LIN {X -0.248,Y -541.721,Z 1405.628,A 0.000,B 0.000,C 90.000,E1 148.997} C_DIS
LIN {X -0.026,Y -544.533,Z 1405.623,A 0.000,B 0.000,C 90.000,E1 148.122} C_DIS
LIN {X 0.196,Y -546.222,Z 1405.620,A 0.000,B 0.000,C 90.000,E1 147.533} C_DIS
LIN {X 0.004,Y -548.398,Z 1405.615,A 0.000,B 0.000,C 90.000,E1 146.707} C_DIS
LIN {X -0.112,Y -550.816,Z 1405.609,A 0.000,B 0.000,C 90.000,E1 145.595} C_DIS
LIN {X -0.256,Y -552.252,Z 1405.604,A 0.000,B 0.000,C 90.000,E1 144.769} C_DIS
LIN {X -0.066,Y -553.322,Z 1405.599,A 0.000,B 0.000,C 90.000,E1 143.909} C_DIS
LIN {X 0.212,Y -554.490,Z 1405.593,A 0.000,B 0.000,C 90.000,E1 142.763} C_DIS
LIN {X 0.069,Y -555.501,Z 1405.587,A 0.000,B 0.000,C 90.000,E1 141.662} C_DIS
LIN {X 0.018,Y -556.739,Z 1405.579,A 0.000,B 0.000,C 90.000,E1 140.275} C_DIS
LIN {X -0.102,Y -557.519,Z 1405.573,A 0.000,B 0.000,C 90.000,E1 139.175} C_DIS
LIN {X -0.196,Y -558.310,Z 1405.565,A 0.000,B 0.000,C 90.000,E1 137.796} C_DIS
LIN {X 0.032,Y -558.832,Z 1405.559,A 0.000,B 0.000,C 90.000,E1 136.662} C_DIS
LIN {X -0.046,Y -559.385,Z 1405.552,A 0.000,B 0.000,C 90.000,E1 135.283} C_DIS
LIN {X -0.192,Y -559.704,Z 1405.545,A 0.000,B 0.000,C 90.000,E1 134.190} C_DIS
LIN {X 0.136,Y -560.065,Z 1405.538,A 0.000,B 0.000,C 90.000,E1 132.771} C_DIS
LIN {X 0.008,Y -560.188,Z 1405.532,A 0.000,B 0.000,C 90.000,E1 131.676} C_DIS
LIN {X 0.139,Y -560.368,Z 1405.521,A 0.000,B 0.000,C 90.000,E1 129.725} C_DIS
LIN {X -0.174,Y -560.676,Z 1405.512,A 0.000,B 0.000,C 90.000,E1 128.096} C_DIS
LIN {X -0.144,Y -560.829,Z 1405.504,A 0.000,B 0.000,C 90.000,E1 126.710} C_DIS
LIN {X 0.003,Y -560.849,Z 1405.496,A 0.000,B 0.000,C 90.000,E1 125.311} C_DIS
LIN {X -0.005,Y -561.268,Z 1405.481,A 0.000,B 0.000,C 90.000,E1 122.546} C_DIS
LIN {X 0.083,Y -561.611,Z 1405.479,A 0.000,B 0.000,C 90.000,E1 122.260} C_DIS
LIN {X -0.232,Y -561.927,Z 1405.477,A 0.000,B 0.000,C 90.000,E1 121.878} C_DIS
LIN {X -0.040,Y -562.328,Z 1405.476,A 0.000,B 0.000,C 90.000,E1 121.720} C_DIS
LIN {X -0.254,Y -563.108,Z 1405.474,A 0.000,B 0.000,C 90.000,E1 121.258} C_DIS
LIN {X 0.206,Y -564.134,Z 1405.472,A 0.000,B 0.000,C 90.000,E1 121.003} C_DIS
LIN {X -0.097,Y -566.068,Z 1405.472,A 0.000,B 0.000,C 90.000,E1 120.924} C_DIS
LIN {X -0.002,Y -567.840,Z 1405.471,A 0.000,B 0.000,C 90.000,E1 120.846} C_DIS
LIN {X 0.227,Y -573.827,Z 1405.471,A 0.000,B 0.000,C 90.000,E1 120.669} C_DIS
LIN {X 0.258,Y -579.247,Z 1405.470,A 0.000,B 0.000,C 90.000,E1 120.590} C_DIS
LIN {X 0.183,Y -581.728,Z 1405.470,A 0.000,B 0.000,C 90.000,E1 120.541} C_DIS
LIN {X 0.143,Y -584.144,Z 1405.469,A 0.000,B 0.000,C 90.000,E1 120.463} C_DIS
LIN {X 0.234,Y -586.696,Z 1405.469,A 0.000,B 0.000,C 90.000,E1 120.335} C_DIS
LIN {X -0.041,Y -589.555,Z 1405.468,A 0.000,B 0.000,C 90.000,E1 120.207} C_DIS
LIN {X 0.287,Y -592.453,Z 1405.467,A 0.000,B 0.000,C 90.000,E1 120.001} C_DIS
LIN {X 0.078,Y -597.897,Z 1405.465,A 0.000,B 0.000,C 90.000,E1 119.617} C_DIS
LIN {X 0.189,Y -603.137,Z 1405.462,A 0.000,B 0.000,C 90.000,E1 119.155} C_DIS
LIN {X -0.118,Y -606.860,Z 1405.460,A 0.000,B 0.000,C 90.000,E1 118.821} C_DIS
LIN {X -0.111,Y -609.008,Z 1405.459,A 0.000,B 0.000,C 90.000,E1 118.565} C_DIS
LIN {X 0.109,Y -612.046,Z 1405.457,A 0.000,B 0.000,C 90.000,E1 118.153} C_DIS
LIN {X 0.041,Y -615.591,Z 1405.454,A 0.000,B 0.000,C 90.000,E1 117.641} C_DIS
LIN {X -0.008,Y -619.104,Z 1405.450,A 0.000,B 0.000,C 90.000,E1 117.001} C_DIS
LIN {X -0.015,Y -619.633,Z 1405.449,A 0.000,B 0.000,C 90.000,E1 116.873} C_DIS
LIN {X -0.036,Y -621.269,Z 1405.445,A 0.000,B 0.000,C 90.000,E1 116.104} C_DIS
LIN {X -0.040,Y -621.342,Z 1405.444,A 0.000,B 0.000,C 90.000,E1 115.848} C_DIS
LIN {X -0.042,Y -621.209,Z 1405.442,A 0.000,B 0.000,C 90.000,E1 115.591} C_DIS
LIN {X -0.044,Y -620.763,Z 1405.441,A 0.000,B 0.000,C 90.000,E1 115.335} C_DIS
LIN {X -0.053,Y -618.848,Z 1405.438,A 0.000,B 0.000,C 90.000,E1 114.823} C_DIS
LIN {X -0.062,Y -616.821,Z 1405.437,A 0.000,B 0.000,C 90.000,E1 114.567} C_DIS
LIN {X 0.030,Y -614.783,Z 1405.435,A 0.000,B 0.000,C 90.000,E1 114.259} C_DIS
LIN {X 0.020,Y -613.342,Z 1405.434,A 0.000,B 0.000,C 90.000,E1 114.131} C_DIS
LIN {X -0.037,Y -606.794,Z 1405.432,A 0.000,B 0.000,C 90.000,E1 113.695} C_DIS
LIN {X 0.065,Y -599.335,Z 1405.430,A 0.000,B 0.000,C 90.000,E1 113.334} C_DIS
LIN {X -0.118,Y -589.005,Z 1405.427,A 0.000,B 0.000,C 90.000,E1 112.950} C_DIS
LIN {X 0.105,Y -585.189,Z 1405.427,A 0.000,B 0.000,C 90.000,E1 112.770} C_DIS
LIN {X 0.059,Y -585.235,Z 1405.427,A 0.000,B 0.000,C 90.000,E1 112.770} C_DIS
LIN {X -0.328,Y -588.195,Z 1405.425,A 0.000,B 0.000,C 90.000,E1 112.589} C_DIS
LIN {X 0.216,Y -595.378,Z 1405.423,A 0.000,B 0.000,C 90.000,E1 112.078} C_DIS
LIN {X -0.256,Y -601.161,Z 1405.421,A 0.000,B 0.000,C 90.000,E1 111.716} C_DIS
LIN {X 0.185,Y -605.437,Z 1405.419,A 0.000,B 0.000,C 90.000,E1 111.354} C_DIS
LIN {X 0.068,Y -610.886,Z 1405.416,A 0.000,B 0.000,C 90.000,E1 110.918} C_DIS
LIN {X 0.296,Y -617.284,Z 1405.413,A 0.000,B 0.000,C 90.000,E1 110.301} C_DIS
LIN {X 0.233,Y -621.031,Z 1405.411,A 0.000,B 0.000,C 90.000,E1 109.939} C_DIS
LIN {X 0.039,Y -625.525,Z 1405.408,A 0.000,B 0.000,C 90.000,E1 109.450} C_DIS
LIN {X -0.190,Y -629.572,Z 1405.405,A 0.000,B 0.000,C 90.000,E1 108.960} C_DIS
LIN {X 0.021,Y -634.903,Z 1405.401,A 0.000,B 0.000,C 90.000,E1 108.181} C_DIS
LIN {X -0.327,Y -638.717,Z 1405.398,A 0.000,B 0.000,C 90.000,E1 107.583} C_DIS
LIN {X -0.030,Y -642.239,Z 1405.393,A 0.000,B 0.000,C 90.000,E1 106.804} C_DIS
LIN {X -0.166,Y -643.953,Z 1405.391,A 0.000,B 0.000,C 90.000,E1 106.315} C_DIS
LIN {X 0.299,Y -644.698,Z 1405.389,A 0.000,B 0.000,C 90.000,E1 106.024} C_DIS
LIN {X 0.003,Y -645.737,Z 1405.386,A 0.000,B 0.000,C 90.000,E1 105.552} C_DIS
LIN {X 0.222,Y -647.242,Z 1405.381,A 0.000,B 0.000,C 90.000,E1 104.537} C_DIS
LIN {X -0.195,Y -648.196,Z 1405.377,A 0.000,B 0.000,C 90.000,E1 103.828} C_DIS
LIN {X 0.027,Y -648.755,Z 1405.373,A 0.000,B 0.000,C 90.000,E1 103.063} C_DIS
LIN {X -0.243,Y -648.886,Z 1405.370,A 0.000,B 0.000,C 90.000,E1 102.591} C_DIS
LIN {X -0.016,Y -648.656,Z 1405.366,A 0.000,B 0.000,C 90.000,E1 101.827} C_DIS
LIN {X 0.343,Y -648.336,Z 1405.363,A 0.000,B 0.000,C 90.000,E1 101.299} C_DIS
LIN {X -0.060,Y -647.747,Z 1405.360,A 0.000,B 0.000,C 90.000,E1 100.838} C_DIS
LIN {X 0.293,Y -646.917,Z 1405.357,A 0.000,B 0.000,C 90.000,E1 100.310} C_DIS
LIN {X -0.259,Y -645.272,Z 1405.353,A 0.000,B 0.000,C 90.000,E1 99.613} C_DIS
LIN {X -0.033,Y -643.887,Z 1405.351,A 0.000,B 0.000,C 90.000,E1 99.095} C_DIS
LIN {X 0.286,Y -642.274,Z 1405.348,A 0.000,B 0.000,C 90.000,E1 98.568} C_DIS
LIN {X -0.140,Y -640.471,Z 1405.345,A 0.000,B 0.000,C 90.000,E1 98.106} C_DIS
LIN {X -0.120,Y -637.221,Z 1405.341,A 0.000,B 0.000,C 90.000,E1 97.352} C_DIS
LIN {X -0.075,Y -634.206,Z 1405.337,A 0.000,B 0.000,C 90.000,E1 96.720} C_DIS
LIN {X 0.080,Y -631.519,Z 1405.335,A 0.000,B 0.000,C 90.000,E1 96.201} C_DIS
LIN {X -0.149,Y -626.443,Z 1405.330,A 0.000,B 0.000,C 90.000,E1 95.334} C_DIS
LIN {X -0.198,Y -622.212,Z 1405.326,A 0.000,B 0.000,C 90.000,E1 94.702} C_DIS
LIN {X -0.176,Y -618.355,Z 1405.323,A 0.000,B 0.000,C 90.000,E1 94.188} C_DIS
LIN {X -0.092,Y -612.452,Z 1405.320,A 0.000,B 0.000,C 90.000,E1 93.555} C_DIS
LIN {X 0.056,Y -604.236,Z 1405.316,A 0.000,B 0.000,C 90.000,E1 92.808} C_DIS
LIN {X -0.056,Y -597.375,Z 1405.313,A 0.000,B 0.000,C 90.000,E1 92.236} C_DIS
LIN {X 0.161,Y -590.138,Z 1405.309,A 0.000,B 0.000,C 90.000,E1 91.661} C_DIS
LIN {X -0.180,Y -581.695,Z 1405.307,A 0.000,B 0.000,C 90.000,E1 91.203} C_DIS
LIN {X -0.243,Y -578.344,Z 1405.306,A 0.000,B 0.000,C 90.000,E1 91.031} C_DIS
LIN {X 0.048,Y -577.150,Z 1405.305,A 0.000,B 0.000,C 90.000,E1 90.917} C_DIS
LIN {X -0.255,Y -576.182,Z 1405.305,A 0.000,B 0.000,C 90.000,E1 90.859} C_DIS
LIN {X -0.076,Y -574.207,Z 1405.304,A 0.000,B 0.000,C 90.000,E1 90.688} C_DIS
LIN {X 0.146,Y -573.809,Z 1405.303,A 0.000,B 0.000,C 90.000,E1 90.573} C_DIS
LIN {X -0.068,Y -573.399,Z 1405.303,A 0.000,B 0.000,C 90.000,E1 90.458} C_DIS
LIN {X -0.139,Y -573.123,Z 1405.300,A 0.000,B 0.000,C 90.000,E1 90.057} C_DIS
LIN {X -0.252,Y -573.569,Z 1405.296,A 0.000,B 0.000,C 90.000,E1 89.255} C_DIS
LIN {X -0.237,Y -574.603,Z 1405.290,A 0.000,B 0.000,C 90.000,E1 88.165} C_DIS
LIN {X 0.097,Y -576.049,Z 1405.281,A 0.000,B 0.000,C 90.000,E1 86.502} C_DIS
LIN {X 0.260,Y -578.153,Z 1405.269,A 0.000,B 0.000,C 90.000,E1 84.318} C_DIS
LIN {X 0.173,Y -579.997,Z 1405.260,A 0.000,B 0.000,C 90.000,E1 82.704} C_DIS
LIN {X 0.081,Y -582.504,Z 1405.248,A 0.000,B 0.000,C 90.000,E1 80.557} C_DIS
LIN {X 0.256,Y -584.296,Z 1405.239,A 0.000,B 0.000,C 90.000,E1 78.926} C_DIS
LIN {X 0.209,Y -585.615,Z 1405.231,A 0.000,B 0.000,C 90.000,E1 77.589} C_DIS
LIN {X -0.209,Y -587.158,Z 1405.221,A 0.000,B 0.000,C 90.000,E1 75.755} C_DIS
LIN {X 0.051,Y -588.113,Z 1405.213,A 0.000,B 0.000,C 90.000,E1 74.393} C_DIS
LIN {X 0.169,Y -588.956,Z 1405.204,A 0.000,B 0.000,C 90.000,E1 72.779} C_DIS
LIN {X 0.057,Y -589.735,Z 1405.197,A 0.000,B 0.000,C 90.000,E1 71.456} C_DIS
LIN {X 0.271,Y -590.290,Z 1405.191,A 0.000,B 0.000,C 90.000,E1 70.369} C_DIS
LIN {X 0.254,Y -591.216,Z 1405.182,A 0.000,B 0.000,C 90.000,E1 68.773} C_DIS
LIN {X -0.293,Y -592.162,Z 1405.173,A 0.000,B 0.000,C 90.000,E1 67.230} C_DIS
LIN {X 0.047,Y -593.134,Z 1405.166,A 0.000,B 0.000,C 90.000,E1 65.869} C_DIS
LIN {X -0.174,Y -594.804,Z 1405.154,A 0.000,B 0.000,C 90.000,E1 63.768} C_DIS
LIN {X -0.003,Y -595.667,Z 1405.148,A 0.000,B 0.000,C 90.000,E1 62.692} C_DIS
LIN {X -0.251,Y -596.932,Z 1405.140,A 0.000,B 0.000,C 90.000,E1 61.129} C_DIS
LIN {X -0.090,Y -598.138,Z 1405.132,A 0.000,B 0.000,C 90.000,E1 59.793} C_DIS
LIN {X 0.245,Y -599.835,Z 1405.122,A 0.000,B 0.000,C 90.000,E1 57.916} C_DIS
LIN {X -0.046,Y -601.029,Z 1405.115,A 0.000,B 0.000,C 90.000,E1 56.628} C_DIS
LIN {X 0.169,Y -602.724,Z 1405.104,A 0.000,B 0.000,C 90.000,E1 54.769} C_DIS
LIN {X 0.015,Y -604.096,Z 1405.096,A 0.000,B 0.000,C 90.000,E1 53.210} C_DIS
LIN {X -0.011,Y -605.038,Z 1405.088,A 0.000,B 0.000,C 90.000,E1 51.904} C_DIS
LIN {X -0.285,Y -605.755,Z 1405.083,A 0.000,B 0.000,C 90.000,E1 50.884} C_DIS
LIN {X 0.097,Y -606.454,Z 1405.075,A 0.000,B 0.000,C 90.000,E1 49.542} C_DIS
LIN {X 0.224,Y -606.791,Z 1405.070,A 0.000,B 0.000,C 90.000,E1 48.485} C_DIS
LIN {X -0.098,Y -606.994,Z 1405.064,A 0.000,B 0.000,C 90.000,E1 47.472} C_DIS
LIN {X 0.253,Y -607.092,Z 1405.057,A 0.000,B 0.000,C 90.000,E1 46.134} C_DIS
LIN {X 0.170,Y -606.960,Z 1405.049,A 0.000,B 0.000,C 90.000,E1 44.838} C_DIS
LIN {X -0.396,Y -606.798,Z 1405.045,A 0.000,B 0.000,C 90.000,E1 44.109} C_DIS
LIN {X -0.049,Y -606.219,Z 1405.038,A 0.000,B 0.000,C 90.000,E1 42.771} C_DIS
LIN {X -0.376,Y -605.679,Z 1405.032,A 0.000,B 0.000,C 90.000,E1 41.757} C_DIS
LIN {X -0.258,Y -604.916,Z 1405.026,A 0.000,B 0.000,C 90.000,E1 40.701} C_DIS
LIN {X -0.151,Y -604.057,Z 1405.020,A 0.000,B 0.000,C 90.000,E1 39.644} C_DIS
LIN {X 0.191,Y -602.658,Z 1405.013,A 0.000,B 0.000,C 90.000,E1 38.302} C_DIS
LIN {X -0.121,Y -601.286,Z 1405.007,A 0.000,B 0.000,C 90.000,E1 37.282} C_DIS
LIN {X 0.028,Y -599.737,Z 1405.001,A 0.000,B 0.000,C 90.000,E1 36.217} C_DIS
LIN {X 0.046,Y -597.330,Z 1404.994,A 0.000,B 0.000,C 90.000,E1 34.898} C_DIS
LIN {X -0.091,Y -595.578,Z 1404.990,A 0.000,B 0.000,C 90.000,E1 34.119} C_DIS
LIN {X 0.136,Y -593.099,Z 1404.984,A 0.000,B 0.000,C 90.000,E1 33.038} C_DIS
LIN {X -0.167,Y -590.165,Z 1404.978,A 0.000,B 0.000,C 90.000,E1 32.005} C_DIS
LIN {X -0.201,Y -587.697,Z 1404.973,A 0.000,B 0.000,C 90.000,E1 31.209} C_DIS
LIN {X 0.039,Y -584.826,Z 1404.969,A 0.000,B 0.000,C 90.000,E1 30.384} C_DIS
LIN {X -0.213,Y -582.703,Z 1404.966,A 0.000,B 0.000,C 90.000,E1 29.873} C_DIS
LIN {X 0.184,Y -579.098,Z 1404.961,A 0.000,B 0.000,C 90.000,E1 29.027} C_DIS
LIN {X 0.029,Y -575.229,Z 1404.957,A 0.000,B 0.000,C 90.000,E1 28.231} C_DIS
LIN {X 0.167,Y -569.424,Z 1404.951,A 0.000,B 0.000,C 90.000,E1 27.129} C_DIS
LIN {X -0.034,Y -563.032,Z 1404.945,A 0.000,B 0.000,C 90.000,E1 26.052} C_DIS
LIN {X 0.128,Y -557.707,Z 1404.940,A 0.000,B 0.000,C 90.000,E1 25.207} C_DIS
LIN {X -0.186,Y -554.901,Z 1404.938,A 0.000,B 0.000,C 90.000,E1 24.823} C_DIS
LIN {X 0.265,Y -549.905,Z 1404.934,A 0.000,B 0.000,C 90.000,E1 24.079} C_DIS
LIN {X -0.089,Y -546.716,Z 1404.932,A 0.000,B 0.000,C 90.000,E1 23.695} C_DIS
LIN {X 0.154,Y -539.977,Z 1404.927,A 0.000,B 0.000,C 90.000,E1 22.823} C_DIS
LIN {X -0.097,Y -535.186,Z 1404.924,A 0.000,B 0.000,C 90.000,E1 22.280} C_DIS
LIN {X -0.121,Y -525.115,Z 1404.917,A 0.000,B 0.000,C 90.000,E1 21.153} C_DIS
LIN {X 0.217,Y -514.660,Z 1404.911,A 0.000,B 0.000,C 90.000,E1 19.993} C_DIS
LIN {X -0.074,Y -503.744,Z 1404.905,A 0.000,B 0.000,C 90.000,E1 18.906} C_DIS
LIN {X 0.113,Y -492.777,Z 1404.899,A 0.000,B 0.000,C 90.000,E1 17.764} C_DIS
LIN {X -0.079,Y -479.251,Z 1404.891,A 0.000,B 0.000,C 90.000,E1 16.386} C_DIS
LIN {X 0.106,Y -465.482,Z 1404.883,A 0.000,B 0.000,C 90.000,E1 14.898} C_DIS
LIN {X 0.055,Y -451.731,Z 1404.875,A 0.000,B 0.000,C 90.000,E1 13.411} C_DIS
LIN {X -0.024,Y -437.847,Z 1404.866,A 0.000,B 0.000,C 90.000,E1 11.883} C_DIS
LIN {X 0.143,Y -417.481,Z 1404.853,A 0.000,B 0.000,C 90.000,E1 9.443} C_DIS
LIN {X -0.048,Y -406.843,Z 1404.845,A 0.000,B 0.000,C 90.000,E1 8.106} C_DIS
LIN {X -0.059,Y -397.404,Z 1404.838,A 0.000,B 0.000,C 90.000,E1 6.891} C_DIS
LIN {X -0.091,Y -393.336,Z 1404.835,A 0.000,B 0.000,C 90.000,E1 6.372} C_DIS
LIN {X -0.063,Y -389.246,Z 1404.832,A 0.000,B 0.000,C 90.000,E1 5.739} C_DIS
LIN {X 0.031,Y -387.720,Z 1404.830,A 0.000,B 0.000,C 90.000,E1 5.391} C_DIS
LIN {X -0.007,Y -387.701,Z 1404.830,A 0.000,B 0.000,C 90.000,E1 5.391} C_DIS
LIN {X -0.180,Y -387.716,Z 1404.829,A 0.000,B 0.000,C 90.000,E1 5.277} C_DIS
LIN {X 0.168,Y -387.721,Z 1404.829,A 0.000,B 0.000,C 90.000,E1 5.220} C_DIS
LIN {X 0.163,Y -389.100,Z 1404.828,A 0.000,B 0.000,C 90.000,E1 4.992} C_DIS
LIN {X -0.132,Y -393.604,Z 1404.825,A 0.000,B 0.000,C 90.000,E1 4.531} C_DIS
LIN {X 0.071,Y -398.766,Z 1404.822,A 0.000,B 0.000,C 90.000,E1 4.012} C_DIS
LIN {X 0.183,Y -403.247,Z 1404.820,A 0.000,B 0.000,C 90.000,E1 3.555} C_DIS
LIN {X 0.078,Y -405.907,Z 1404.818,A 0.000,B 0.000,C 90.000,E1 3.269} C_DIS
LIN {X -0.134,Y -410.707,Z 1404.815,A 0.000,B 0.000,C 90.000,E1 2.694} C_DIS
LIN {X -0.107,Y -416.714,Z 1404.810,A 0.000,B 0.000,C 90.000,E1 1.835} C_DIS
LIN {X -0.025,Y -422.984,Z 1404.804,A 0.000,B 0.000,C 90.000,E1 0.802} C_DIS
LIN {X 0.000,Y -427.486,Z 1404.800,A 0.000,B 0.000,C 90.000,E1 360.000} C_DIS
LIN {X -0.203,Y -430.023,Z 1404.797,A 0.000,B 0.000,C 90.000,E1 359.484} C_DIS
LIN {X -0.131,Y -431.361,Z 1404.795,A 0.000,B 0.000,C 90.000,E1 359.141} C_DIS
LIN {X -0.054,Y -432.419,Z 1404.793,A 0.000,B 0.000,C 90.000,E1 358.797} C_DIS
LIN {X 0.025,Y -433.006,Z 1404.792,A 0.000,B 0.000,C 90.000,E1 358.453} C_DIS
LIN {X 0.121,Y -432.563,Z 1404.790,A 0.000,B 0.000,C 90.000,E1 358.108} C_DIS
LIN {X -0.129,Y -431.791,Z 1404.789,A 0.000,B 0.000,C 90.000,E1 358.051} C_DIS
LIN {X -0.009,Y -430.732,Z 1404.789,A 0.000,B 0.000,C 90.000,E1 357.993} C_DIS
LIN {X 0.095,Y -360.544,Z 1404.787,A 0.000,B 0.000,C 90.000,E1 357.593} C_DIS
LIN {X 0.063,Y -359.781,Z 1404.787,A 0.000,B 0.000,C 90.000,E1 357.593} C_DIS
LIN {X 0.049,Y -359.377,Z 1404.768,A 0.000,B 0.000,C 90.000,E1 354.204} C_DIS
LIN {X -0.057,Y -359.540,Z 1404.726,A 0.000,B 0.000,C 90.000,E1 346.700} C_DIS
LIN {X -0.101,Y -361.978,Z 1404.682,A 0.000,B 0.000,C 90.000,E1 338.827} C_DIS
LIN {X 0.007,Y -365.931,Z 1404.643,A 0.000,B 0.000,C 90.000,E1 331.719} C_DIS
LIN {X -0.235,Y -366.221,Z 1404.641,A 0.000,B 0.000,C 90.000,E1 331.385} C_DIS
LIN {X -0.017,Y -371.299,Z 1404.604,A 0.000,B 0.000,C 90.000,E1 324.689} C_DIS
LIN {X -0.029,Y -371.726,Z 1404.602,A 0.000,B 0.000,C 90.000,E1 324.322} C_DIS
LIN {X 0.051,Y -377.296,Z 1404.567,A 0.000,B 0.000,C 90.000,E1 318.081} C_DIS
LIN {X -0.204,Y -378.205,Z 1404.563,A 0.000,B 0.000,C 90.000,E1 317.391} C_DIS
LIN {X 0.068,Y -383.875,Z 1404.531,A 0.000,B 0.000,C 90.000,E1 311.553} C_DIS
LIN {X 0.117,Y -384.853,Z 1404.527,A 0.000,B 0.000,C 90.000,E1 310.825} C_DIS
LIN {X 0.039,Y -390.546,Z 1404.495,A 0.000,B 0.000,C 90.000,E1 305.105} C_DIS
LIN {X 0.106,Y -391.038,Z 1404.493,A 0.000,B 0.000,C 90.000,E1 304.739} C_DIS
LIN {X -0.048,Y -391.401,Z 1404.491,A 0.000,B 0.000,C 90.000,E1 304.405} C_DIS
LIN {X -0.105,Y -396.764,Z 1404.460,A 0.000,B 0.000,C 90.000,E1 298.743} C_DIS
LIN {X 0.114,Y -397.099,Z 1404.458,A 0.000,B 0.000,C 90.000,E1 298.359} C_DIS
LIN {X -0.101,Y -401.554,Z 1404.427,A 0.000,B 0.000,C 90.000,E1 292.770} C_DIS
LIN {X 0.042,Y -404.617,Z 1404.396,A 0.000,B 0.000,C 90.000,E1 287.166} C_DIS
LIN {X 0.144,Y -404.756,Z 1404.394,A 0.000,B 0.000,C 90.000,E1 286.804} C_DIS
LIN {X 0.142,Y -406.072,Z 1404.365,A 0.000,B 0.000,C 90.000,E1 281.591} C_DIS
LIN {X 0.151,Y -406.113,Z 1404.363,A 0.000,B 0.000,C 90.000,E1 281.243} C_DIS
LIN {X -0.218,Y -405.669,Z 1404.334,A 0.000,B 0.000,C 90.000,E1 276.087} C_DIS
LIN {X 0.191,Y -405.559,Z 1404.332,A 0.000,B 0.000,C 90.000,E1 275.682} C_DIS
LIN {X -0.138,Y -403.525,Z 1404.305,A 0.000,B 0.000,C 90.000,E1 270.859} C_DIS
LIN {X -0.171,Y -403.316,Z 1404.303,A 0.000,B 0.000,C 90.000,E1 270.516} C_DIS
LIN {X 0.018,Y -398.973,Z 1404.272,A 0.000,B 0.000,C 90.000,E1 264.894} C_DIS
LIN {X -0.176,Y -393.145,Z 1404.242,A 0.000,B 0.000,C 90.000,E1 259.634} C_DIS
LIN {X -0.144,Y -392.879,Z 1404.240,A 0.000,B 0.000,C 90.000,E1 259.275} C_DIS
LIN {X -0.121,Y -386.043,Z 1404.213,A 0.000,B 0.000,C 90.000,E1 254.283} C_DIS
LIN {X -0.075,Y -385.314,Z 1404.209,A 0.000,B 0.000,C 90.000,E1 253.559} C_DIS
LIN {X -0.053,Y -384.856,Z 1404.207,A 0.000,B 0.000,C 90.000,E1 253.196} C_DIS
LIN {X 0.049,Y -378.034,Z 1404.183,A 0.000,B 0.000,C 90.000,E1 248.847} C_DIS
LIN {X -0.074,Y -376.287,Z 1404.174,A 0.000,B 0.000,C 90.000,E1 247.411} C_DIS
LIN {X -0.095,Y -375.734,Z 1404.172,A 0.000,B 0.000,C 90.000,E1 247.050} C_DIS
LIN {X 0.009,Y -368.995,Z 1404.150,A 0.000,B 0.000,C 90.000,E1 242.999} C_DIS
LIN {X -0.088,Y -366.137,Z 1404.138,A 0.000,B 0.000,C 90.000,E1 240.795} C_DIS
LIN {X -0.182,Y -359.266,Z 1404.115,A 0.000,B 0.000,C 90.000,E1 236.707} C_DIS
LIN {X 0.044,Y -355.929,Z 1404.100,A 0.000,B 0.000,C 90.000,E1 234.036} C_DIS
LIN {X 0.135,Y -348.858,Z 1404.075,A 0.000,B 0.000,C 90.000,E1 229.461} C_DIS
LIN {X -0.025,Y -346.236,Z 1404.062,A 0.000,B 0.000,C 90.000,E1 227.187} C_DIS
LIN {X 0.098,Y -345.767,Z 1404.060,A 0.000,B 0.000,C 90.000,E1 226.782} C_DIS
LIN {X 0.058,Y -339.037,Z 1404.032,A 0.000,B 0.000,C 90.000,E1 221.757} C_DIS
LIN {X -0.077,Y -336.890,Z 1404.019,A 0.000,B 0.000,C 90.000,E1 219.439} C_DIS
LIN {X -0.060,Y -331.224,Z 1403.991,A 0.000,B 0.000,C 90.000,E1 214.326} C_DIS
LIN {X -0.002,Y -329.324,Z 1403.975,A 0.000,B 0.000,C 90.000,E1 211.544} C_DIS
LIN {X 0.102,Y -326.741,Z 1403.960,A 0.000,B 0.000,C 90.000,E1 208.743} C_DIS
LIN {X 0.049,Y -323.850,Z 1403.929,A 0.000,B 0.000,C 90.000,E1 203.153} C_DIS
LIN {X -0.029,Y -321.117,Z 1403.882,A 0.000,B 0.000,C 90.000,E1 194.717} C_DIS
LIN {X 0.126,Y -320.949,Z 1403.877,A 0.000,B 0.000,C 90.000,E1 193.883} C_DIS
LIN {X -0.095,Y -321.537,Z 1403.833,A 0.000,B 0.000,C 90.000,E1 185.853} C_DIS
LIN {X 0.058,Y -321.880,Z 1403.818,A 0.000,B 0.000,C 90.000,E1 183.212} C_DIS
LIN {X 0.041,Y -322.010,Z 1403.818,A 0.000,B 0.000,C 90.000,E1 183.212} C_DIS
LIN {X -0.076,Y -380.157,Z 1403.815,A 0.000,B 0.000,C 90.000,E1 182.751} C_DIS
LIN {X -0.036,Y -404.490,Z 1403.814,A 0.000,B 0.000,C 90.000,E1 182.579} C_DIS
LIN {X 0.056,Y -405.380,Z 1403.814,A 0.000,B 0.000,C 90.000,E1 182.522} C_DIS
LIN {X 0.048,Y -406.415,Z 1403.813,A 0.000,B 0.000,C 90.000,E1 182.350} C_DIS
LIN {X 0.023,Y -406.681,Z 1403.811,A 0.000,B 0.000,C 90.000,E1 182.007} C_DIS
LIN {X 0.013,Y -406.227,Z 1403.809,A 0.000,B 0.000,C 90.000,E1 181.661} C_DIS
LIN {X -0.009,Y -405.444,Z 1403.807,A 0.000,B 0.000,C 90.000,E1 181.318} C_DIS
LIN {X -0.085,Y -402.271,Z 1403.802,A 0.000,B 0.000,C 90.000,E1 180.286} C_DIS
LIN {X -0.176,Y -399.329,Z 1403.797,A 0.000,B 0.000,C 90.000,E1 179.427} C_DIS
LIN {X 0.065,Y -395.105,Z 1403.791,A 0.000,B 0.000,C 90.000,E1 178.339} C_DIS
LIN {X -0.055,Y -391.954,Z 1403.787,A 0.000,B 0.000,C 90.000,E1 177.650} C_DIS
LIN {X 0.102,Y -386.517,Z 1403.781,A 0.000,B 0.000,C 90.000,E1 176.560} C_DIS
LIN {X -0.007,Y -382.305,Z 1403.777,A 0.000,B 0.000,C 90.000,E1 175.869} C_DIS
LIN {X -0.113,Y -379.215,Z 1403.774,A 0.000,B 0.000,C 90.000,E1 175.355} C_DIS
LIN {X 0.025,Y -375.001,Z 1403.770,A 0.000,B 0.000,C 90.000,E1 174.609} C_DIS
LIN {X -0.136,Y -367.360,Z 1403.762,A 0.000,B 0.000,C 90.000,E1 173.166} C_DIS
LIN {X -0.003,Y -360.265,Z 1403.754,A 0.000,B 0.000,C 90.000,E1 171.659} C_DIS
LIN {X -0.096,Y -356.457,Z 1403.749,A 0.000,B 0.000,C 90.000,E1 170.735} C_DIS
LIN {X 0.197,Y -355.789,Z 1403.747,A 0.000,B 0.000,C 90.000,E1 170.500} C_DIS
LIN {X 0.074,Y -353.844,Z 1403.743,A 0.000,B 0.000,C 90.000,E1 169.634} C_DIS
LIN {X 0.056,Y -353.847,Z 1403.743,A 0.000,B 0.000,C 90.000,E1 169.634} C_DIS
LIN {X 0.050,Y -354.052,Z 1403.741,A 0.000,B 0.000,C 90.000,E1 169.454} C_DIS
LIN {X 0.031,Y -354.068,Z 1403.741,A 0.000,B 0.000,C 90.000,E1 169.454} C_DIS
LIN {X 0.152,Y -356.199,Z 1403.739,A 0.000,B 0.000,C 90.000,E1 168.993} C_DIS
LIN {X 0.094,Y -357.279,Z 1403.738,A 0.000,B 0.000,C 90.000,E1 168.814} C_DIS
LIN {X 0.087,Y -363.769,Z 1403.733,A 0.000,B 0.000,C 90.000,E1 167.881} C_DIS
LIN {X -0.125,Y -370.956,Z 1403.728,A 0.000,B 0.000,C 90.000,E1 166.992} C_DIS
LIN {X 0.110,Y -381.370,Z 1403.721,A 0.000,B 0.000,C 90.000,E1 165.755} C_DIS
LIN {X 0.108,Y -395.004,Z 1403.713,A 0.000,B 0.000,C 90.000,E1 164.338} C_DIS
LIN {X -0.227,Y -408.989,Z 1403.706,A 0.000,B 0.000,C 90.000,E1 163.087} C_DIS
LIN {X 0.040,Y -429.378,Z 1403.696,A 0.000,B 0.000,C 90.000,E1 161.348} C_DIS
LIN {X -0.101,Y -441.821,Z 1403.691,A 0.000,B 0.000,C 90.000,E1 160.369} C_DIS
LIN {X 0.102,Y -452.731,Z 1403.686,A 0.000,B 0.000,C 90.000,E1 159.464} C_DIS
LIN {X -0.007,Y -461.853,Z 1403.682,A 0.000,B 0.000,C 90.000,E1 158.720} C_DIS
LIN {X -0.205,Y -470.920,Z 1403.678,A 0.000,B 0.000,C 90.000,E1 157.975} C_DIS
LIN {X -0.015,Y -478.217,Z 1403.674,A 0.000,B 0.000,C 90.000,E1 157.305} C_DIS
LIN {X 0.104,Y -488.340,Z 1403.669,A 0.000,B 0.000,C 90.000,E1 156.357} C_DIS
LIN {X 0.185,Y -496.794,Z 1403.664,A 0.000,B 0.000,C 90.000,E1 155.537} C_DIS
LIN {X 0.296,Y -502.222,Z 1403.661,A 0.000,B 0.000,C 90.000,E1 154.973} C_DIS
LIN {X 0.087,Y -508.823,Z 1403.657,A 0.000,B 0.000,C 90.000,E1 154.280} C_DIS
LIN {X -0.030,Y -515.154,Z 1403.653,A 0.000,B 0.000,C 90.000,E1 153.563} C_DIS
LIN {X -0.084,Y -518.751,Z 1403.651,A 0.000,B 0.000,C 90.000,E1 153.127} C_DIS
LIN {X -0.002,Y -523.136,Z 1403.647,A 0.000,B 0.000,C 90.000,E1 152.538} C_DIS
LIN {X -0.131,Y -527.174,Z 1403.644,A 0.000,B 0.000,C 90.000,E1 151.975} C_DIS
LIN {X -0.031,Y -530.831,Z 1403.641,A 0.000,B 0.000,C 90.000,E1 151.385} C_DIS
LIN {X 0.098,Y -534.049,Z 1403.638,A 0.000,B 0.000,C 90.000,E1 150.795} C_DIS
LIN {X 0.109,Y -537.416,Z 1403.634,A 0.000,B 0.000,C 90.000,E1 150.078} C_DIS
LIN {X -0.179,Y -539.809,Z 1403.631,A 0.000,B 0.000,C 90.000,E1 149.537} C_DIS
LIN {X 0.010,Y -541.911,Z 1403.628,A 0.000,B 0.000,C 90.000,E1 148.948} C_DIS
LIN {X -0.232,Y -544.700,Z 1403.623,A 0.000,B 0.000,C 90.000,E1 148.122} C_DIS
LIN {X -0.009,Y -546.379,Z 1403.620,A 0.000,B 0.000,C 90.000,E1 147.533} C_DIS
LIN {X 0.060,Y -547.868,Z 1403.617,A 0.000,B 0.000,C 90.000,E1 146.962} C_DIS
LIN {X -0.059,Y -550.338,Z 1403.610,A 0.000,B 0.000,C 90.000,E1 145.849} C_DIS
LIN {X 0.192,Y -551.393,Z 1403.607,A 0.000,B 0.000,C 90.000,E1 145.261} C_DIS
LIN {X 0.310,Y -552.314,Z 1403.604,A 0.000,B 0.000,C 90.000,E1 144.689} C_DIS
LIN {X -0.268,Y -553.344,Z 1403.599,A 0.000,B 0.000,C 90.000,E1 143.909} C_DIS
LIN {X 0.010,Y -554.498,Z 1403.593,A 0.000,B 0.000,C 90.000,E1 142.763} C_DIS
LIN {X -0.134,Y -555.489,Z 1403.587,A 0.000,B 0.000,C 90.000,E1 141.662} C_DIS
LIN {X -0.185,Y -556.717,Z 1403.579,A 0.000,B 0.000,C 90.000,E1 140.275} C_DIS
LIN {X 0.058,Y -557.484,Z 1403.573,A 0.000,B 0.000,C 90.000,E1 139.138} C_DIS
LIN {X -0.025,Y -558.262,Z 1403.565,A 0.000,B 0.000,C 90.000,E1 137.757} C_DIS
LIN {X 0.233,Y -558.748,Z 1403.559,A 0.000,B 0.000,C 90.000,E1 136.620} C_DIS
LIN {X 0.140,Y -559.314,Z 1403.552,A 0.000,B 0.000,C 90.000,E1 135.243} C_DIS
LIN {X 0.058,Y -559.702,Z 1403.544,A 0.000,B 0.000,C 90.000,E1 133.866} C_DIS
LIN {X 0.005,Y -560.026,Z 1403.536,A 0.000,B 0.000,C 90.000,E1 132.486} C_DIS
LIN {X -0.119,Y -560.139,Z 1403.530,A 0.000,B 0.000,C 90.000,E1 131.391} C_DIS
LIN {X -0.324,Y -560.425,Z 1403.518,A 0.000,B 0.000,C 90.000,E1 129.197} C_DIS
LIN {X -0.293,Y -560.707,Z 1403.510,A 0.000,B 0.000,C 90.000,E1 127.810} C_DIS
LIN {X 0.187,Y -560.809,Z 1403.502,A 0.000,B 0.000,C 90.000,E1 126.377} C_DIS
LIN {X -0.023,Y -560.888,Z 1403.493,A 0.000,B 0.000,C 90.000,E1 124.739} C_DIS
LIN {X -0.186,Y -561.175,Z 1403.485,A 0.000,B 0.000,C 90.000,E1 123.372} C_DIS
LIN {X -0.095,Y -561.428,Z 1403.484,A 0.000,B 0.000,C 90.000,E1 123.086} C_DIS
LIN {X -0.218,Y -561.738,Z 1403.481,A 0.000,B 0.000,C 90.000,E1 122.546} C_DIS
LIN {X -0.128,Y -562.199,Z 1403.479,A 0.000,B 0.000,C 90.000,E1 122.260} C_DIS
LIN {X 0.139,Y -562.468,Z 1403.478,A 0.000,B 0.000,C 90.000,E1 121.957} C_DIS
LIN {X 0.231,Y -563.252,Z 1403.476,A 0.000,B 0.000,C 90.000,E1 121.671} C_DIS
LIN {X 0.189,Y -563.270,Z 1403.476,A 0.000,B 0.000,C 90.000,E1 121.671} C_DIS
LIN {X 0.130,Y -564.468,Z 1403.475,A 0.000,B 0.000,C 90.000,E1 121.544} C_DIS
LIN {X 0.227,Y -565.518,Z 1403.475,A 0.000,B 0.000,C 90.000,E1 121.465} C_DIS
LIN {X 0.243,Y -568.853,Z 1403.474,A 0.000,B 0.000,C 90.000,E1 121.337} C_DIS
LIN {X -0.327,Y -570.783,Z 1403.474,A 0.000,B 0.000,C 90.000,E1 121.337} C_DIS
LIN {X -0.064,Y -573.396,Z 1403.474,A 0.000,B 0.000,C 90.000,E1 121.258} C_DIS
LIN {X -0.099,Y -576.908,Z 1403.473,A 0.000,B 0.000,C 90.000,E1 121.209} C_DIS
LIN {X 0.182,Y -582.660,Z 1403.473,A 0.000,B 0.000,C 90.000,E1 121.052} C_DIS
LIN {X -0.210,Y -584.830,Z 1403.472,A 0.000,B 0.000,C 90.000,E1 121.003} C_DIS
LIN {X 0.181,Y -590.764,Z 1403.471,A 0.000,B 0.000,C 90.000,E1 120.669} C_DIS
LIN {X -0.239,Y -593.494,Z 1403.470,A 0.000,B 0.000,C 90.000,E1 120.541} C_DIS
LIN {X 0.164,Y -597.643,Z 1403.468,A 0.000,B 0.000,C 90.000,E1 120.207} C_DIS
LIN {X 0.106,Y -600.461,Z 1403.467,A 0.000,B 0.000,C 90.000,E1 120.001} C_DIS
LIN {X 0.128,Y -605.765,Z 1403.464,A 0.000,B 0.000,C 90.000,E1 119.539} C_DIS
LIN {X -0.265,Y -609.392,Z 1403.462,A 0.000,B 0.000,C 90.000,E1 119.205} C_DIS
LIN {X -0.270,Y -613.674,Z 1403.459,A 0.000,B 0.000,C 90.000,E1 118.693} C_DIS
LIN {X -0.022,Y -616.436,Z 1403.457,A 0.000,B 0.000,C 90.000,E1 118.281} C_DIS
LIN {X -0.054,Y -618.969,Z 1403.455,A 0.000,B 0.000,C 90.000,E1 117.897} C_DIS
LIN {X -0.072,Y -621.333,Z 1403.453,A 0.000,B 0.000,C 90.000,E1 117.513} C_DIS
LIN {X -0.076,Y -621.998,Z 1403.452,A 0.000,B 0.000,C 90.000,E1 117.385} C_DIS
LIN {X -0.073,Y -624.883,Z 1403.448,A 0.000,B 0.000,C 90.000,E1 116.616} C_DIS
LIN {X -0.054,Y -625.502,Z 1403.445,A 0.000,B 0.000,C 90.000,E1 116.104} C_DIS
LIN {X -0.042,Y -625.654,Z 1403.444,A 0.000,B 0.000,C 90.000,E1 115.848} C_DIS
LIN {X -0.018,Y -625.252,Z 1403.441,A 0.000,B 0.000,C 90.000,E1 115.335} C_DIS
LIN {X -0.007,Y -624.484,Z 1403.439,A 0.000,B 0.000,C 90.000,E1 115.079} C_DIS
LIN {X 0.006,Y -622.753,Z 1403.437,A 0.000,B 0.000,C 90.000,E1 114.695} C_DIS
LIN {X -0.249,Y -621.995,Z 1403.437,A 0.000,B 0.000,C 90.000,E1 114.591} C_DIS
LIN {X -0.246,Y -619.313,Z 1403.435,A 0.000,B 0.000,C 90.000,E1 114.335} C_DIS
LIN {X -0.095,Y -617.345,Z 1403.434,A 0.000,B 0.000,C 90.000,E1 114.079} C_DIS
LIN {X -0.108,Y -613.326,Z 1403.432,A 0.000,B 0.000,C 90.000,E1 113.823} C_DIS
LIN {X -0.183,Y -610.441,Z 1403.431,A 0.000,B 0.000,C 90.000,E1 113.643} C_DIS
LIN {X 0.091,Y -608.295,Z 1403.431,A 0.000,B 0.000,C 90.000,E1 113.515} C_DIS
LIN {X 0.106,Y -606.564,Z 1403.430,A 0.000,B 0.000,C 90.000,E1 113.462} C_DIS
LIN {X 0.362,Y -605.392,Z 1403.430,A 0.000,B 0.000,C 90.000,E1 113.387} C_DIS
LIN {X -0.188,Y -601.954,Z 1403.429,A 0.000,B 0.000,C 90.000,E1 113.259} C_DIS
LIN {X 0.026,Y -595.632,Z 1403.428,A 0.000,B 0.000,C 90.000,E1 113.025} C_DIS
LIN {X -0.235,Y -588.915,Z 1403.426,A 0.000,B 0.000,C 90.000,E1 112.770} C_DIS
LIN {X -0.280,Y -588.946,Z 1403.426,A 0.000,B 0.000,C 90.000,E1 112.770} C_DIS
LIN {X 0.186,Y -591.331,Z 1403.425,A 0.000,B 0.000,C 90.000,E1 112.514} C_DIS
LIN {X 0.045,Y -596.206,Z 1403.423,A 0.000,B 0.000,C 90.000,E1 112.206} C_DIS
LIN {X 0.282,Y -602.039,Z 1403.421,A 0.000,B 0.000,C 90.000,E1 111.770} C_DIS
LIN {X 0.140,Y -606.377,Z 1403.419,A 0.000,B 0.000,C 90.000,E1 111.461} C_DIS
LIN {X -0.178,Y -611.839,Z 1403.417,A 0.000,B 0.000,C 90.000,E1 111.046} C_DIS
LIN {X 0.028,Y -616.975,Z 1403.414,A 0.000,B 0.000,C 90.000,E1 110.556} C_DIS
LIN {X 0.073,Y -621.959,Z 1403.412,A 0.000,B 0.000,C 90.000,E1 110.066} C_DIS
LIN {X -0.099,Y -626.482,Z 1403.409,A 0.000,B 0.000,C 90.000,E1 109.577} C_DIS
LIN {X -0.321,Y -630.605,Z 1403.406,A 0.000,B 0.000,C 90.000,E1 109.087} C_DIS
LIN {X -0.109,Y -635.895,Z 1403.402,A 0.000,B 0.000,C 90.000,E1 108.308} C_DIS
LIN {X 0.166,Y -640.439,Z 1403.397,A 0.000,B 0.000,C 90.000,E1 107.528} C_DIS
LIN {X 0.040,Y -643.399,Z 1403.394,A 0.000,B 0.000,C 90.000,E1 106.913} C_DIS
LIN {X -0.118,Y -644.384,Z 1403.393,A 0.000,B 0.000,C 90.000,E1 106.677} C_DIS
LIN {X 0.198,Y -646.004,Z 1403.390,A 0.000,B 0.000,C 90.000,E1 106.150} C_DIS
LIN {X -0.056,Y -647.581,Z 1403.386,A 0.000,B 0.000,C 90.000,E1 105.426} C_DIS
LIN {X 0.047,Y -649.372,Z 1403.379,A 0.000,B 0.000,C 90.000,E1 104.175} C_DIS
LIN {X -0.222,Y -649.933,Z 1403.376,A 0.000,B 0.000,C 90.000,E1 103.703} C_DIS
LIN {X 0.013,Y -650.373,Z 1403.372,A 0.000,B 0.000,C 90.000,E1 102.939} C_DIS
LIN {X 0.385,Y -650.451,Z 1403.369,A 0.000,B 0.000,C 90.000,E1 102.411} C_DIS
LIN {X -0.144,Y -650.127,Z 1403.365,A 0.000,B 0.000,C 90.000,E1 101.715} C_DIS
LIN {X -0.276,Y -649.983,Z 1403.364,A 0.000,B 0.000,C 90.000,E1 101.478} C_DIS
LIN {X -0.042,Y -649.056,Z 1403.359,A 0.000,B 0.000,C 90.000,E1 100.715} C_DIS
LIN {X 0.201,Y -648.212,Z 1403.357,A 0.000,B 0.000,C 90.000,E1 100.197} C_DIS
LIN {X -0.083,Y -647.126,Z 1403.354,A 0.000,B 0.000,C 90.000,E1 99.726} C_DIS
LIN {X 0.003,Y -645.030,Z 1403.350,A 0.000,B 0.000,C 90.000,E1 98.973} C_DIS
LIN {X 0.067,Y -642.495,Z 1403.346,A 0.000,B 0.000,C 90.000,E1 98.219} C_DIS
LIN {X -0.188,Y -641.570,Z 1403.344,A 0.000,B 0.000,C 90.000,E1 97.992} C_DIS
LIN {X -0.155,Y -638.257,Z 1403.340,A 0.000,B 0.000,C 90.000,E1 97.239} C_DIS
LIN {X 0.032,Y -635.833,Z 1403.337,A 0.000,B 0.000,C 90.000,E1 96.720} C_DIS
LIN {X 0.199,Y -633.176,Z 1403.335,A 0.000,B 0.000,C 90.000,E1 96.201} C_DIS
LIN {X -0.013,Y -628.094,Z 1403.330,A 0.000,B 0.000,C 90.000,E1 95.334} C_DIS
LIN {X -0.049,Y -623.985,Z 1403.326,A 0.000,B 0.000,C 90.000,E1 94.702} C_DIS
LIN {X -0.016,Y -620.178,Z 1403.323,A 0.000,B 0.000,C 90.000,E1 94.188} C_DIS
LIN {X 0.190,Y -616.749,Z 1403.321,A 0.000,B 0.000,C 90.000,E1 93.784} C_DIS
LIN {X -0.104,Y -614.327,Z 1403.320,A 0.000,B 0.000,C 90.000,E1 93.555} C_DIS
LIN {X 0.112,Y -607.610,Z 1403.316,A 0.000,B 0.000,C 90.000,E1 92.922} C_DIS
LIN {X -0.095,Y -599.342,Z 1403.312,A 0.000,B 0.000,C 90.000,E1 92.236} C_DIS
LIN {X -0.099,Y -595.048,Z 1403.311,A 0.000,B 0.000,C 90.000,E1 91.892} C_DIS
LIN {X 0.026,Y -590.581,Z 1403.309,A 0.000,B 0.000,C 90.000,E1 91.547} C_DIS
LIN {X 0.036,Y -583.791,Z 1403.306,A 0.000,B 0.000,C 90.000,E1 91.146} C_DIS
LIN {X -0.098,Y -577.273,Z 1403.304,A 0.000,B 0.000,C 90.000,E1 90.802} C_DIS
LIN {X -0.104,Y -575.649,Z 1403.304,A 0.000,B 0.000,C 90.000,E1 90.688} C_DIS
LIN {X 0.202,Y -573.906,Z 1403.303,A 0.000,B 0.000,C 90.000,E1 90.458} C_DIS
LIN {X -0.145,Y -573.519,Z 1403.302,A 0.000,B 0.000,C 90.000,E1 90.344} C_DIS
LIN {X 0.169,Y -573.223,Z 1403.300,A 0.000,B 0.000,C 90.000,E1 90.000} C_DIS
LIN {X -0.119,Y -573.382,Z 1403.297,A 0.000,B 0.000,C 90.000,E1 89.484} C_DIS
LIN {X 0.185,Y -574.849,Z 1403.288,A 0.000,B 0.000,C 90.000,E1 87.822} C_DIS
LIN {X -0.056,Y -576.267,Z 1403.279,A 0.000,B 0.000,C 90.000,E1 86.216} C_DIS
LIN {X -0.041,Y -578.156,Z 1403.268,A 0.000,B 0.000,C 90.000,E1 84.318} C_DIS
LIN {X -0.129,Y -580.008,Z 1403.259,A 0.000,B 0.000,C 90.000,E1 82.704} C_DIS
LIN {X -0.221,Y -582.514,Z 1403.247,A 0.000,B 0.000,C 90.000,E1 80.557} C_DIS
LIN {X -0.048,Y -584.312,Z 1403.239,A 0.000,B 0.000,C 90.000,E1 78.926} C_DIS
LIN {X -0.095,Y -585.617,Z 1403.231,A 0.000,B 0.000,C 90.000,E1 77.589} C_DIS
LIN {X -0.192,Y -586.921,Z 1403.222,A 0.000,B 0.000,C 90.000,E1 75.992} C_DIS
LIN {X -0.017,Y -587.554,Z 1403.218,A 0.000,B 0.000,C 90.000,E1 75.172} C_DIS
LIN {X -0.007,Y -588.258,Z 1403.212,A 0.000,B 0.000,C 90.000,E1 74.102} C_DIS
LIN {X 0.107,Y -589.122,Z 1403.203,A 0.000,B 0.000,C 90.000,E1 72.489} C_DIS
LIN {X 0.180,Y -589.905,Z 1403.195,A 0.000,B 0.000,C 90.000,E1 71.148} C_DIS
LIN {X 0.074,Y -590.602,Z 1403.188,A 0.000,B 0.000,C 90.000,E1 69.826} C_DIS
LIN {X -0.163,Y -591.378,Z 1403.181,A 0.000,B 0.000,C 90.000,E1 68.518} C_DIS
LIN {X 0.281,Y -592.036,Z 1403.175,A 0.000,B 0.000,C 90.000,E1 67.411} C_DIS
LIN {X -0.015,Y -593.163,Z 1403.166,A 0.000,B 0.000,C 90.000,E1 65.845} C_DIS
LIN {X 0.054,Y -594.836,Z 1403.154,A 0.000,B 0.000,C 90.000,E1 63.717} C_DIS
LIN {X -0.035,Y -595.701,Z 1403.148,A 0.000,B 0.000,C 90.000,E1 62.666} C_DIS
LIN {X 0.255,Y -596.963,Z 1403.139,A 0.000,B 0.000,C 90.000,E1 61.051} C_DIS
LIN {X 0.122,Y -598.171,Z 1403.132,A 0.000,B 0.000,C 90.000,E1 59.744} C_DIS
LIN {X -0.059,Y -599.882,Z 1403.122,A 0.000,B 0.000,C 90.000,E1 57.916} C_DIS
LIN {X -0.108,Y -601.314,Z 1403.113,A 0.000,B 0.000,C 90.000,E1 56.342} C_DIS
LIN {X 0.117,Y -602.992,Z 1403.103,A 0.000,B 0.000,C 90.000,E1 54.482} C_DIS
LIN {X -0.289,Y -604.145,Z 1403.095,A 0.000,B 0.000,C 90.000,E1 53.210} C_DIS
LIN {X -0.315,Y -605.099,Z 1403.088,A 0.000,B 0.000,C 90.000,E1 51.904} C_DIS
LIN {X 0.264,Y -605.815,Z 1403.082,A 0.000,B 0.000,C 90.000,E1 50.803} C_DIS
LIN {X -0.207,Y -606.513,Z 1403.075,A 0.000,B 0.000,C 90.000,E1 49.542} C_DIS
LIN {X -0.078,Y -606.843,Z 1403.069,A 0.000,B 0.000,C 90.000,E1 48.485} C_DIS
LIN {X -0.399,Y -607.048,Z 1403.064,A 0.000,B 0.000,C 90.000,E1 47.472} C_DIS
LIN {X -0.048,Y -607.141,Z 1403.056,A 0.000,B 0.000,C 90.000,E1 46.134} C_DIS
LIN {X -0.130,Y -606.997,Z 1403.049,A 0.000,B 0.000,C 90.000,E1 44.838} C_DIS
LIN {X 0.163,Y -606.830,Z 1403.045,A 0.000,B 0.000,C 90.000,E1 44.028} C_DIS
LIN {X 0.317,Y -606.116,Z 1403.036,A 0.000,B 0.000,C 90.000,E1 42.447} C_DIS
LIN {X -0.016,Y -605.524,Z 1403.030,A 0.000,B 0.000,C 90.000,E1 41.434} C_DIS
LIN {X 0.353,Y -604.561,Z 1403.023,A 0.000,B 0.000,C 90.000,E1 40.092} C_DIS
LIN {X 0.019,Y -604.122,Z 1403.020,A 0.000,B 0.000,C 90.000,E1 39.600} C_DIS
LIN {X -0.103,Y -602.723,Z 1403.013,A 0.000,B 0.000,C 90.000,E1 38.302} C_DIS
LIN {X 0.065,Y -601.378,Z 1403.007,A 0.000,B 0.000,C 90.000,E1 37.237} C_DIS
LIN {X 0.221,Y -599.826,Z 1403.001,A 0.000,B 0.000,C 90.000,E1 36.171} C_DIS
LIN {X -0.134,Y -597.908,Z 1402.995,A 0.000,B 0.000,C 90.000,E1 35.152} C_DIS
LIN {X 0.223,Y -596.302,Z 1402.991,A 0.000,B 0.000,C 90.000,E1 34.326} C_DIS
LIN {X -0.147,Y -593.204,Z 1402.984,A 0.000,B 0.000,C 90.000,E1 33.038} C_DIS
LIN {X 0.053,Y -590.278,Z 1402.978,A 0.000,B 0.000,C 90.000,E1 31.957} C_DIS
LIN {X 0.328,Y -587.822,Z 1402.973,A 0.000,B 0.000,C 90.000,E1 31.131} C_DIS
LIN {X 0.269,Y -584.932,Z 1402.969,A 0.000,B 0.000,C 90.000,E1 30.335} C_DIS
LIN {X 0.310,Y -582.807,Z 1402.966,A 0.000,B 0.000,C 90.000,E1 29.795} C_DIS
LIN {X 0.124,Y -578.591,Z 1402.961,A 0.000,B 0.000,C 90.000,E1 28.871} C_DIS
LIN {X -0.315,Y -574.588,Z 1402.956,A 0.000,B 0.000,C 90.000,E1 28.103} C_DIS
LIN {X -0.097,Y -569.526,Z 1402.951,A 0.000,B 0.000,C 90.000,E1 27.129} C_DIS
LIN {X -0.046,Y -563.116,Z 1402.945,A 0.000,B 0.000,C 90.000,E1 26.027} C_DIS
LIN {X -0.128,Y -557.832,Z 1402.940,A 0.000,B 0.000,C 90.000,E1 25.207} C_DIS
LIN {X 0.064,Y -555.014,Z 1402.938,A 0.000,B 0.000,C 90.000,E1 24.771} C_DIS
LIN {X -0.102,Y -548.995,Z 1402.933,A 0.000,B 0.000,C 90.000,E1 23.951} C_DIS
LIN {X 0.186,Y -542.342,Z 1402.928,A 0.000,B 0.000,C 90.000,E1 23.078} C_DIS
LIN {X 0.022,Y -536.512,Z 1402.924,A 0.000,B 0.000,C 90.000,E1 22.386} C_DIS
LIN {X -0.174,Y -526.524,Z 1402.918,A 0.000,B 0.000,C 90.000,E1 21.280} C_DIS
LIN {X 0.138,Y -516.161,Z 1402.912,A 0.000,B 0.000,C 90.000,E1 20.120} C_DIS
LIN {X -0.173,Y -505.261,Z 1402.906,A 0.000,B 0.000,C 90.000,E1 19.033} C_DIS
LIN {X -0.067,Y -492.903,Z 1402.899,A 0.000,B 0.000,C 90.000,E1 17.764} C_DIS
LIN {X -0.029,Y -477.904,Z 1402.890,A 0.000,B 0.000,C 90.000,E1 16.205} C_DIS
LIN {X -0.004,Y -462.778,Z 1402.881,A 0.000,B 0.000,C 90.000,E1 14.592} C_DIS
LIN {X -0.002,Y -447.509,Z 1402.872,A 0.000,B 0.000,C 90.000,E1 12.939} C_DIS
LIN {X -0.174,Y -437.757,Z 1402.866,A 0.000,B 0.000,C 90.000,E1 11.883} C_DIS
LIN {X -0.107,Y -416.308,Z 1402.852,A 0.000,B 0.000,C 90.000,E1 9.321} C_DIS
LIN {X 0.082,Y -405.653,Z 1402.844,A 0.000,B 0.000,C 90.000,E1 7.936} C_DIS
LIN {X 0.165,Y -396.247,Z 1402.838,A 0.000,B 0.000,C 90.000,E1 6.720} C_DIS
LIN {X 0.165,Y -393.543,Z 1402.836,A 0.000,B 0.000,C 90.000,E1 6.372} C_DIS
LIN {X -0.128,Y -389.483,Z 1402.832,A 0.000,B 0.000,C 90.000,E1 5.796} C_DIS
LIN {X -0.035,Y -388.114,Z 1402.830,A 0.000,B 0.000,C 90.000,E1 5.454} C_DIS
LIN {X -0.073,Y -388.097,Z 1402.830,A 0.000,B 0.000,C 90.000,E1 5.454} C_DIS
LIN {X -0.048,Y -388.262,Z 1402.829,A 0.000,B 0.000,C 90.000,E1 5.277} C_DIS
LIN {X -0.086,Y -388.275,Z 1402.829,A 0.000,B 0.000,C 90.000,E1 5.277} C_DIS
LIN {X -0.145,Y -389.104,Z 1402.829,A 0.000,B 0.000,C 90.000,E1 5.163} C_DIS
LIN {X 0.039,Y -392.863,Z 1402.826,A 0.000,B 0.000,C 90.000,E1 4.702} C_DIS
LIN {X -0.040,Y -399.762,Z 1402.823,A 0.000,B 0.000,C 90.000,E1 4.073} C_DIS
LIN {X 0.103,Y -404.346,Z 1402.820,A 0.000,B 0.000,C 90.000,E1 3.612} C_DIS
LIN {X 0.064,Y -411.056,Z 1402.816,A 0.000,B 0.000,C 90.000,E1 2.808} C_DIS
LIN {X 0.142,Y -418.266,Z 1402.810,A 0.000,B 0.000,C 90.000,E1 1.776} C_DIS
LIN {X -0.191,Y -424.602,Z 1402.804,A 0.000,B 0.000,C 90.000,E1 0.802} C_DIS
LIN {X 0.000,Y -429.297,Z 1402.800,A 0.000,B 0.000,C 90.000,E1 360.000} C_DIS
LIN {X -0.157,Y -433.228,Z 1402.796,A 0.000,B 0.000,C 90.000,E1 359.312} C_DIS
LIN {X -0.029,Y -435.605,Z 1402.793,A 0.000,B 0.000,C 90.000,E1 358.797} C_DIS
LIN {X 0.065,Y -436.994,Z 1402.792,A 0.000,B 0.000,C 90.000,E1 358.453} C_DIS
LIN {X 0.179,Y -438.178,Z 1402.790,A 0.000,B 0.000,C 90.000,E1 358.108} C_DIS
LIN {X -0.157,Y -438.957,Z 1402.788,A 0.000,B 0.000,C 90.000,E1 357.822} C_DIS
LIN {X -0.049,Y -439.142,Z 1402.786,A 0.000,B 0.000,C 90.000,E1 357.478} C_DIS
LIN {X 0.005,Y -438.683,Z 1402.785,A 0.000,B 0.000,C 90.000,E1 357.306} C_DIS
LIN {X -0.186,Y -438.003,Z 1402.785,A 0.000,B 0.000,C 90.000,E1 357.249} C_DIS
LIN {X -0.063,Y -437.161,Z 1402.784,A 0.000,B 0.000,C 90.000,E1 357.192} C_DIS
LIN {X 0.154,Y -359.818,Z 1402.781,A 0.000,B 0.000,C 90.000,E1 356.560} C_DIS
LIN {X 0.134,Y -359.545,Z 1402.781,A 0.000,B 0.000,C 90.000,E1 356.560} C_DIS
LIN {X 0.167,Y -359.408,Z 1402.768,A 0.000,B 0.000,C 90.000,E1 354.261} C_DIS
LIN {X 0.068,Y -359.507,Z 1402.727,A 0.000,B 0.000,C 90.000,E1 346.756} C_DIS
LIN {X 0.151,Y -359.542,Z 1402.722,A 0.000,B 0.000,C 90.000,E1 345.992} C_DIS
LIN {X -0.092,Y -361.964,Z 1402.683,A 0.000,B 0.000,C 90.000,E1 338.901} C_DIS
LIN {X -0.077,Y -366.192,Z 1402.641,A 0.000,B 0.000,C 90.000,E1 331.435} C_DIS
LIN {X -0.053,Y -371.213,Z 1402.604,A 0.000,B 0.000,C 90.000,E1 324.769} C_DIS
LIN {X -0.065,Y -371.645,Z 1402.602,A 0.000,B 0.000,C 90.000,E1 324.402} C_DIS
LIN {X -0.010,Y -376.750,Z 1402.570,A 0.000,B 0.000,C 90.000,E1 318.528} C_DIS
LIN {X 0.002,Y -378.145,Z 1402.564,A 0.000,B 0.000,C 90.000,E1 317.433} C_DIS
LIN {X 0.020,Y -384.267,Z 1402.529,A 0.000,B 0.000,C 90.000,E1 311.272} C_DIS
LIN {X 0.062,Y -384.770,Z 1402.527,A 0.000,B 0.000,C 90.000,E1 310.906} C_DIS
LIN {X 0.052,Y -390.938,Z 1402.494,A 0.000,B 0.000,C 90.000,E1 304.818} C_DIS
LIN {X -0.102,Y -391.359,Z 1402.492,A 0.000,B 0.000,C 90.000,E1 304.485} C_DIS
LIN {X 0.069,Y -397.068,Z 1402.458,A 0.000,B 0.000,C 90.000,E1 298.437} C_DIS
LIN {X 0.024,Y -401.473,Z 1402.427,A 0.000,B 0.000,C 90.000,E1 292.823} C_DIS
LIN {X -0.182,Y -401.765,Z 1402.423,A 0.000,B 0.000,C 90.000,E1 292.153} C_DIS
LIN {X 0.151,Y -404.555,Z 1402.396,A 0.000,B 0.000,C 90.000,E1 287.221} C_DIS
LIN {X -0.135,Y -404.761,Z 1402.394,A 0.000,B 0.000,C 90.000,E1 286.913} C_DIS
LIN {X 0.159,Y -406.032,Z 1402.365,A 0.000,B 0.000,C 90.000,E1 281.658} C_DIS
LIN {X -0.229,Y -406.142,Z 1402.363,A 0.000,B 0.000,C 90.000,E1 281.366} C_DIS
LIN {X -0.125,Y -405.653,Z 1402.334,A 0.000,B 0.000,C 90.000,E1 276.144} C_DIS
LIN {X -0.120,Y -405.610,Z 1402.332,A 0.000,B 0.000,C 90.000,E1 275.796} C_DIS
LIN {X -0.047,Y -403.552,Z 1402.305,A 0.000,B 0.000,C 90.000,E1 270.917} C_DIS
LIN {X -0.111,Y -403.054,Z 1402.301,A 0.000,B 0.000,C 90.000,E1 270.229} C_DIS
LIN {X 0.113,Y -399.015,Z 1402.272,A 0.000,B 0.000,C 90.000,E1 264.951} C_DIS
LIN {X 0.007,Y -397.648,Z 1402.266,A 0.000,B 0.000,C 90.000,E1 263.913} C_DIS
LIN {X -0.112,Y -392.932,Z 1402.241,A 0.000,B 0.000,C 90.000,E1 259.342} C_DIS
LIN {X -0.154,Y -392.475,Z 1402.239,A 0.000,B 0.000,C 90.000,E1 258.993} C_DIS
LIN {X -0.006,Y -386.120,Z 1402.213,A 0.000,B 0.000,C 90.000,E1 254.338} C_DIS
LIN {X -0.046,Y -384.988,Z 1402.207,A 0.000,B 0.000,C 90.000,E1 253.268} C_DIS
LIN {X 0.181,Y -378.129,Z 1402.183,A 0.000,B 0.000,C 90.000,E1 248.901} C_DIS
LIN {X -0.084,Y -376.369,Z 1402.175,A 0.000,B 0.000,C 90.000,E1 247.486} C_DIS
LIN {X 0.041,Y -375.876,Z 1402.173,A 0.000,B 0.000,C 90.000,E1 247.102} C_DIS
LIN {X -0.008,Y -369.101,Z 1402.151,A 0.000,B 0.000,C 90.000,E1 243.076} C_DIS
LIN {X 0.071,Y -366.252,Z 1402.138,A 0.000,B 0.000,C 90.000,E1 240.845} C_DIS
LIN {X 0.032,Y -358.848,Z 1402.113,A 0.000,B 0.000,C 90.000,E1 236.373} C_DIS
LIN {X 0.020,Y -356.038,Z 1402.101,A 0.000,B 0.000,C 90.000,E1 234.116} C_DIS
LIN {X 0.016,Y -348.475,Z 1402.073,A 0.000,B 0.000,C 90.000,E1 229.175} C_DIS
LIN {X 0.077,Y -345.893,Z 1402.060,A 0.000,B 0.000,C 90.000,E1 226.863} C_DIS
LIN {X 0.044,Y -339.120,Z 1402.032,A 0.000,B 0.000,C 90.000,E1 221.838} C_DIS
LIN {X 0.128,Y -336.954,Z 1402.020,A 0.000,B 0.000,C 90.000,E1 219.483} C_DIS
LIN {X 0.051,Y -332.754,Z 1402.000,A 0.000,B 0.000,C 90.000,E1 215.964} C_DIS
LIN {X 0.178,Y -329.368,Z 1401.976,A 0.000,B 0.000,C 90.000,E1 211.592} C_DIS
LIN {X 0.190,Y -328.644,Z 1401.971,A 0.000,B 0.000,C 90.000,E1 210.797} C_DIS
LIN {X 0.102,Y -324.091,Z 1401.934,A 0.000,B 0.000,C 90.000,E1 204.027} C_DIS
LIN {X -0.089,Y -323.869,Z 1401.929,A 0.000,B 0.000,C 90.000,E1 203.259} C_DIS
LIN {X 0.085,Y -323.114,Z 1401.922,A 0.000,B 0.000,C 90.000,E1 202.025} C_DIS
LIN {X -0.118,Y -321.123,Z 1401.880,A 0.000,B 0.000,C 90.000,E1 194.411} C_DIS
LIN {X 0.041,Y -321.498,Z 1401.833,A 0.000,B 0.000,C 90.000,E1 185.910} C_DIS
LIN {X 0.040,Y -321.637,Z 1401.826,A 0.000,B 0.000,C 90.000,E1 184.702} C_DIS
LIN {X -0.033,Y -321.675,Z 1401.824,A 0.000,B 0.000,C 90.000,E1 184.359} C_DIS
LIN {X -0.050,Y -321.875,Z 1401.824,A 0.000,B 0.000,C 90.000,E1 184.359} C_DIS
LIN {X -0.043,Y -372.230,Z 1401.821,A 0.000,B 0.000,C 90.000,E1 183.784} C_DIS
LIN {X -0.202,Y -406.157,Z 1401.819,A 0.000,B 0.000,C 90.000,E1 183.498} C_DIS
LIN {X -0.111,Y -409.763,Z 1401.819,A 0.000,B 0.000,C 90.000,E1 183.440} C_DIS
LIN {X -0.087,Y -410.505,Z 1401.819,A 0.000,B 0.000,C 90.000,E1 183.383} C_DIS
LIN {X -0.129,Y -411.534,Z 1401.818,A 0.000,B 0.000,C 90.000,E1 183.151} C_DIS
LIN {X -0.137,Y -411.679,Z 1401.816,A 0.000,B 0.000,C 90.000,E1 182.808} C_DIS
LIN {X -0.141,Y -411.200,Z 1401.814,A 0.000,B 0.000,C 90.000,E1 182.465} C_DIS
LIN {X -0.132,Y -409.567,Z 1401.810,A 0.000,B 0.000,C 90.000,E1 181.776} C_DIS
LIN {X -0.147,Y -407.818,Z 1401.806,A 0.000,B 0.000,C 90.000,E1 181.088} C_DIS
LIN {X -0.174,Y -405.763,Z 1401.802,A 0.000,B 0.000,C 90.000,E1 180.401} C_DIS
LIN {X 0.159,Y -402.253,Z 1401.796,A 0.000,B 0.000,C 90.000,E1 179.312} C_DIS
LIN {X 0.061,Y -398.944,Z 1401.792,A 0.000,B 0.000,C 90.000,E1 178.453} C_DIS
LIN {X -0.060,Y -395.121,Z 1401.787,A 0.000,B 0.000,C 90.000,E1 177.593} C_DIS
LIN {X 0.137,Y -389.626,Z 1401.781,A 0.000,B 0.000,C 90.000,E1 176.502} C_DIS
LIN {X -0.043,Y -382.360,Z 1401.774,A 0.000,B 0.000,C 90.000,E1 175.298} C_DIS
LIN {X 0.019,Y -376.015,Z 1401.768,A 0.000,B 0.000,C 90.000,E1 174.204} C_DIS
LIN {X -0.035,Y -369.270,Z 1401.761,A 0.000,B 0.000,C 90.000,E1 172.932} C_DIS
LIN {X -0.078,Y -360.455,Z 1401.750,A 0.000,B 0.000,C 90.000,E1 171.084} C_DIS
LIN {X 0.059,Y -358.280,Z 1401.747,A 0.000,B 0.000,C 90.000,E1 170.500} C_DIS
LIN {X 0.121,Y -356.519,Z 1401.744,A 0.000,B 0.000,C 90.000,E1 169.926} C_DIS
LIN {X 0.009,Y -355.679,Z 1401.742,A 0.000,B 0.000,C 90.000,E1 169.567} C_DIS
LIN {X 0.051,Y -355.336,Z 1401.741,A 0.000,B 0.000,C 90.000,E1 169.342} C_DIS
LIN {X 0.033,Y -355.337,Z 1401.741,A 0.000,B 0.000,C 90.000,E1 169.342} C_DIS
LIN {X 0.051,Y -356.851,Z 1401.739,A 0.000,B 0.000,C 90.000,E1 168.993} C_DIS
LIN {X -0.008,Y -357.842,Z 1401.738,A 0.000,B 0.000,C 90.000,E1 168.814} C_DIS
LIN {X 0.121,Y -361.386,Z 1401.735,A 0.000,B 0.000,C 90.000,E1 168.229} C_DIS
LIN {X 0.108,Y -368.290,Z 1401.730,A 0.000,B 0.000,C 90.000,E1 167.297} C_DIS
LIN {X 0.173,Y -377.129,Z 1401.724,A 0.000,B 0.000,C 90.000,E1 166.228} C_DIS
LIN {X 0.077,Y -392.188,Z 1401.715,A 0.000,B 0.000,C 90.000,E1 164.629} C_DIS
LIN {X -0.116,Y -403.017,Z 1401.709,A 0.000,B 0.000,C 90.000,E1 163.614} C_DIS
LIN {X 0.067,Y -417.044,Z 1401.702,A 0.000,B 0.000,C 90.000,E1 162.362} C_DIS
LIN {X -0.104,Y -434.391,Z 1401.694,A 0.000,B 0.000,C 90.000,E1 160.967} C_DIS
LIN {X 0.119,Y -443.822,Z 1401.690,A 0.000,B 0.000,C 90.000,E1 160.188} C_DIS
LIN {X -0.074,Y -454.682,Z 1401.685,A 0.000,B 0.000,C 90.000,E1 159.337} C_DIS
LIN {X -0.104,Y -465.239,Z 1401.680,A 0.000,B 0.000,C 90.000,E1 158.465} C_DIS
LIN {X 0.140,Y -472.721,Z 1401.677,A 0.000,B 0.000,C 90.000,E1 157.794} C_DIS
LIN {X -0.184,Y -480.004,Z 1401.673,A 0.000,B 0.000,C 90.000,E1 157.177} C_DIS
LIN {X -0.126,Y -490.095,Z 1401.668,A 0.000,B 0.000,C 90.000,E1 156.230} C_DIS
LIN {X -0.011,Y -498.453,Z 1401.663,A 0.000,B 0.000,C 90.000,E1 155.409} C_DIS
LIN {X -0.006,Y -505.036,Z 1401.660,A 0.000,B 0.000,C 90.000,E1 154.717} C_DIS
LIN {X 0.156,Y -511.537,Z 1401.656,A 0.000,B 0.000,C 90.000,E1 153.973} C_DIS
LIN {X -0.086,Y -515.286,Z 1401.653,A 0.000,B 0.000,C 90.000,E1 153.563} C_DIS
LIN {X -0.139,Y -518.836,Z 1401.651,A 0.000,B 0.000,C 90.000,E1 153.127} C_DIS
LIN {X -0.103,Y -523.291,Z 1401.647,A 0.000,B 0.000,C 90.000,E1 152.538} C_DIS
LIN {X -0.120,Y -526.411,Z 1401.645,A 0.000,B 0.000,C 90.000,E1 152.103} C_DIS
LIN {X -0.026,Y -530.157,Z 1401.642,A 0.000,B 0.000,C 90.000,E1 151.513} C_DIS
LIN {X -0.047,Y -534.228,Z 1401.638,A 0.000,B 0.000,C 90.000,E1 150.795} C_DIS
LIN {X 0.107,Y -536.980,Z 1401.635,A 0.000,B 0.000,C 90.000,E1 150.205} C_DIS
LIN {X -0.323,Y -539.963,Z 1401.631,A 0.000,B 0.000,C 90.000,E1 149.537} C_DIS
LIN {X -0.133,Y -542.066,Z 1401.627,A 0.000,B 0.000,C 90.000,E1 148.948} C_DIS
LIN {X 0.089,Y -544.839,Z 1401.623,A 0.000,B 0.000,C 90.000,E1 148.074} C_DIS
LIN {X -0.151,Y -546.511,Z 1401.620,A 0.000,B 0.000,C 90.000,E1 147.533} C_DIS
LIN {X -0.081,Y -547.970,Z 1401.616,A 0.000,B 0.000,C 90.000,E1 146.962} C_DIS
LIN {X 0.257,Y -550.418,Z 1401.610,A 0.000,B 0.000,C 90.000,E1 145.801} C_DIS
LIN {X 0.111,Y -551.918,Z 1401.606,A 0.000,B 0.000,C 90.000,E1 144.975} C_DIS
LIN {X 0.234,Y -552.719,Z 1401.602,A 0.000,B 0.000,C 90.000,E1 144.402} C_DIS
LIN {X 0.173,Y -553.945,Z 1401.596,A 0.000,B 0.000,C 90.000,E1 143.290} C_DIS
LIN {X 0.015,Y -554.999,Z 1401.590,A 0.000,B 0.000,C 90.000,E1 142.190} C_DIS
LIN {X 0.102,Y -556.676,Z 1401.579,A 0.000,B 0.000,C 90.000,E1 140.231} C_DIS
LIN {X 0.263,Y -557.294,Z 1401.575,A 0.000,B 0.000,C 90.000,E1 139.380} C_DIS
LIN {X -0.168,Y -558.197,Z 1401.565,A 0.000,B 0.000,C 90.000,E1 137.757} C_DIS
LIN {X -0.247,Y -558.771,Z 1401.558,A 0.000,B 0.000,C 90.000,E1 136.377} C_DIS
LIN {X 0.057,Y -559.311,Z 1401.550,A 0.000,B 0.000,C 90.000,E1 134.960} C_DIS
LIN {X -0.017,Y -559.697,Z 1401.542,A 0.000,B 0.000,C 90.000,E1 133.581} C_DIS
LIN {X -0.099,Y -559.998,Z 1401.534,A 0.000,B 0.000,C 90.000,E1 132.204} C_DIS
LIN {X -0.065,Y -560.141,Z 1401.525,A 0.000,B 0.000,C 90.000,E1 130.539} C_DIS
LIN {X 0.061,Y -560.503,Z 1401.514,A 0.000,B 0.000,C 90.000,E1 128.588} C_DIS
LIN {X 0.341,Y -560.712,Z 1401.510,A 0.000,B 0.000,C 90.000,E1 127.729} C_DIS
LIN {X 0.131,Y -560.791,Z 1401.501,A 0.000,B 0.000,C 90.000,E1 126.091} C_DIS
LIN {X -0.120,Y -561.241,Z 1401.487,A 0.000,B 0.000,C 90.000,E1 123.627} C_DIS
LIN {X 0.317,Y -561.903,Z 1401.482,A 0.000,B 0.000,C 90.000,E1 122.752} C_DIS
LIN {X 0.075,Y -562.475,Z 1401.480,A 0.000,B 0.000,C 90.000,E1 122.467} C_DIS
LIN {X 0.327,Y -563.230,Z 1401.480,A 0.000,B 0.000,C 90.000,E1 122.339} C_DIS
LIN {X 0.046,Y -564.297,Z 1401.479,A 0.000,B 0.000,C 90.000,E1 122.163} C_DIS
LIN {X -0.164,Y -564.488,Z 1401.479,A 0.000,B 0.000,C 90.000,E1 122.133} C_DIS
LIN {X 0.044,Y -567.356,Z 1401.478,A 0.000,B 0.000,C 90.000,E1 121.957} C_DIS
LIN {X -0.053,Y -569.790,Z 1401.477,A 0.000,B 0.000,C 90.000,E1 121.878} C_DIS
LIN {X -0.149,Y -572.807,Z 1401.477,A 0.000,B 0.000,C 90.000,E1 121.799} C_DIS
LIN {X 0.088,Y -578.695,Z 1401.476,A 0.000,B 0.000,C 90.000,E1 121.671} C_DIS
LIN {X 0.301,Y -581.196,Z 1401.476,A 0.000,B 0.000,C 90.000,E1 121.592} C_DIS
LIN {X -0.042,Y -586.802,Z 1401.475,A 0.000,B 0.000,C 90.000,E1 121.416} C_DIS
LIN {X -0.128,Y -592.587,Z 1401.473,A 0.000,B 0.000,C 90.000,E1 121.131} C_DIS
LIN {X 0.010,Y -598.119,Z 1401.471,A 0.000,B 0.000,C 90.000,E1 120.747} C_DIS
LIN {X -0.278,Y -602.301,Z 1401.469,A 0.000,B 0.000,C 90.000,E1 120.463} C_DIS
LIN {X 0.051,Y -604.804,Z 1401.468,A 0.000,B 0.000,C 90.000,E1 120.207} C_DIS
LIN {X -0.239,Y -608.543,Z 1401.466,A 0.000,B 0.000,C 90.000,E1 119.873} C_DIS
LIN {X 0.172,Y -612.249,Z 1401.464,A 0.000,B 0.000,C 90.000,E1 119.461} C_DIS
LIN {X 0.217,Y -616.400,Z 1401.461,A 0.000,B 0.000,C 90.000,E1 118.949} C_DIS
LIN {X 0.173,Y -620.959,Z 1401.457,A 0.000,B 0.000,C 90.000,E1 118.309} C_DIS
LIN {X -0.382,Y -624.165,Z 1401.455,A 0.000,B 0.000,C 90.000,E1 117.847} C_DIS
LIN {X -0.078,Y -626.646,Z 1401.452,A 0.000,B 0.000,C 90.000,E1 117.308} C_DIS
LIN {X -0.066,Y -627.661,Z 1401.450,A 0.000,B 0.000,C 90.000,E1 117.052} C_DIS
LIN {X -0.031,Y -628.913,Z 1401.448,A 0.000,B 0.000,C 90.000,E1 116.539} C_DIS
LIN {X -0.010,Y -629.318,Z 1401.446,A 0.000,B 0.000,C 90.000,E1 116.283} C_DIS
LIN {X 0.013,Y -629.590,Z 1401.445,A 0.000,B 0.000,C 90.000,E1 116.027} C_DIS
LIN {X 0.037,Y -629.662,Z 1401.443,A 0.000,B 0.000,C 90.000,E1 115.771} C_DIS
LIN {X -0.182,Y -628.849,Z 1401.440,A 0.000,B 0.000,C 90.000,E1 115.283} C_DIS
LIN {X -0.157,Y -628.234,Z 1401.439,A 0.000,B 0.000,C 90.000,E1 115.027} C_DIS
LIN {X -0.125,Y -626.163,Z 1401.437,A 0.000,B 0.000,C 90.000,E1 114.643} C_DIS
LIN {X -0.116,Y -625.566,Z 1401.436,A 0.000,B 0.000,C 90.000,E1 114.515} C_DIS
LIN {X -0.109,Y -624.523,Z 1401.435,A 0.000,B 0.000,C 90.000,E1 114.387} C_DIS
LIN {X -0.014,Y -621.983,Z 1401.434,A 0.000,B 0.000,C 90.000,E1 114.131} C_DIS
LIN {X -0.179,Y -620.971,Z 1401.433,A 0.000,B 0.000,C 90.000,E1 114.027} C_DIS
LIN {X -0.179,Y -619.643,Z 1401.433,A 0.000,B 0.000,C 90.000,E1 113.898} C_DIS
LIN {X -0.306,Y -612.519,Z 1401.431,A 0.000,B 0.000,C 90.000,E1 113.515} C_DIS
LIN {X 0.139,Y -610.644,Z 1401.430,A 0.000,B 0.000,C 90.000,E1 113.387} C_DIS
LIN {X -0.112,Y -608.041,Z 1401.430,A 0.000,B 0.000,C 90.000,E1 113.334} C_DIS
LIN {X -0.120,Y -606.078,Z 1401.429,A 0.000,B 0.000,C 90.000,E1 113.259} C_DIS
LIN {X -0.021,Y -604.412,Z 1401.429,A 0.000,B 0.000,C 90.000,E1 113.153} C_DIS
LIN {X 0.072,Y -601.308,Z 1401.428,A 0.000,B 0.000,C 90.000,E1 113.025} C_DIS
LIN {X 0.037,Y -596.757,Z 1401.427,A 0.000,B 0.000,C 90.000,E1 112.898} C_DIS
LIN {X -0.046,Y -591.885,Z 1401.426,A 0.000,B 0.000,C 90.000,E1 112.695} C_DIS
LIN {X -0.081,Y -591.877,Z 1401.426,A 0.000,B 0.000,C 90.000,E1 112.695} C_DIS
LIN {X -0.114,Y -591.879,Z 1401.426,A 0.000,B 0.000,C 90.000,E1 112.695} C_DIS
LIN {X -0.171,Y -591.899,Z 1401.426,A 0.000,B 0.000,C 90.000,E1 112.695} C_DIS
LIN {X -0.085,Y -594.220,Z 1401.425,A 0.000,B 0.000,C 90.000,E1 112.514} C_DIS
LIN {X -0.036,Y -601.150,Z 1401.422,A 0.000,B 0.000,C 90.000,E1 112.025} C_DIS
LIN {X 0.093,Y -606.861,Z 1401.420,A 0.000,B 0.000,C 90.000,E1 111.589} C_DIS
LIN {X -0.043,Y -613.625,Z 1401.417,A 0.000,B 0.000,C 90.000,E1 111.046} C_DIS
LIN {X 0.187,Y -618.682,Z 1401.414,A 0.000,B 0.000,C 90.000,E1 110.556} C_DIS
LIN {X 0.195,Y -623.621,Z 1401.412,A 0.000,B 0.000,C 90.000,E1 110.066} C_DIS
LIN {X 0.053,Y -627.037,Z 1401.410,A 0.000,B 0.000,C 90.000,E1 109.704} C_DIS
LIN {X -0.119,Y -632.101,Z 1401.406,A 0.000,B 0.000,C 90.000,E1 109.087} C_DIS
LIN {X 0.304,Y -636.527,Z 1401.402,A 0.000,B 0.000,C 90.000,E1 108.417} C_DIS
LIN {X -0.054,Y -639.710,Z 1401.400,A 0.000,B 0.000,C 90.000,E1 107.946} C_DIS
LIN {X -0.194,Y -642.538,Z 1401.397,A 0.000,B 0.000,C 90.000,E1 107.457} C_DIS
LIN {X 0.277,Y -644.287,Z 1401.395,A 0.000,B 0.000,C 90.000,E1 107.040} C_DIS
LIN {X 0.122,Y -645.344,Z 1401.393,A 0.000,B 0.000,C 90.000,E1 106.804} C_DIS
LIN {X 0.008,Y -647.041,Z 1401.391,A 0.000,B 0.000,C 90.000,E1 106.315} C_DIS
LIN {X -0.137,Y -647.787,Z 1401.389,A 0.000,B 0.000,C 90.000,E1 106.079} C_DIS
LIN {X 0.072,Y -649.247,Z 1401.385,A 0.000,B 0.000,C 90.000,E1 105.315} C_DIS
LIN {X -0.291,Y -650.670,Z 1401.380,A 0.000,B 0.000,C 90.000,E1 104.356} C_DIS
LIN {X -0.045,Y -651.485,Z 1401.375,A 0.000,B 0.000,C 90.000,E1 103.592} C_DIS
LIN {X -0.299,Y -651.836,Z 1401.373,A 0.000,B 0.000,C 90.000,E1 103.119} C_DIS
LIN {X 0.085,Y -651.915,Z 1401.370,A 0.000,B 0.000,C 90.000,E1 102.591} C_DIS
LIN {X 0.342,Y -651.642,Z 1401.366,A 0.000,B 0.000,C 90.000,E1 101.827} C_DIS
LIN {X -0.044,Y -651.301,Z 1401.363,A 0.000,B 0.000,C 90.000,E1 101.366} C_DIS
LIN {X 0.205,Y -650.322,Z 1401.359,A 0.000,B 0.000,C 90.000,E1 100.602} C_DIS
LIN {X -0.179,Y -649.436,Z 1401.356,A 0.000,B 0.000,C 90.000,E1 100.141} C_DIS
LIN {X 0.185,Y -648.309,Z 1401.354,A 0.000,B 0.000,C 90.000,E1 99.613} C_DIS
LIN {X -0.208,Y -646.956,Z 1401.351,A 0.000,B 0.000,C 90.000,E1 99.151} C_DIS
LIN {X 0.132,Y -645.366,Z 1401.348,A 0.000,B 0.000,C 90.000,E1 98.624} C_DIS
LIN {X 0.198,Y -642.626,Z 1401.344,A 0.000,B 0.000,C 90.000,E1 97.871} C_DIS
LIN {X 0.155,Y -639.313,Z 1401.340,A 0.000,B 0.000,C 90.000,E1 97.125} C_DIS
LIN {X -0.155,Y -637.472,Z 1401.338,A 0.000,B 0.000,C 90.000,E1 96.777} C_DIS
LIN {X -0.108,Y -634.147,Z 1401.334,A 0.000,B 0.000,C 90.000,E1 96.144} C_DIS
LIN {X 0.320,Y -629.040,Z 1401.329,A 0.000,B 0.000,C 90.000,E1 95.220} C_DIS
LIN {X 0.291,Y -624.889,Z 1401.326,A 0.000,B 0.000,C 90.000,E1 94.588} C_DIS
LIN {X -0.291,Y -621.079,Z 1401.323,A 0.000,B 0.000,C 90.000,E1 94.131} C_DIS
LIN {X -0.228,Y -616.442,Z 1401.320,A 0.000,B 0.000,C 90.000,E1 93.612} C_DIS
LIN {X -0.104,Y -609.835,Z 1401.317,A 0.000,B 0.000,C 90.000,E1 92.980} C_DIS
LIN {X -0.251,Y -601.722,Z 1401.313,A 0.000,B 0.000,C 90.000,E1 92.293} C_DIS
LIN {X -0.286,Y -596.068,Z 1401.310,A 0.000,B 0.000,C 90.000,E1 91.833} C_DIS
LIN {X -0.171,Y -591.521,Z 1401.308,A 0.000,B 0.000,C 90.000,E1 91.489} C_DIS
LIN {X -0.075,Y -589.981,Z 1401.308,A 0.000,B 0.000,C 90.000,E1 91.375} C_DIS
LIN {X -0.110,Y -584.924,Z 1401.306,A 0.000,B 0.000,C 90.000,E1 91.088} C_DIS
LIN {X -0.116,Y -578.390,Z 1401.304,A 0.000,B 0.000,C 90.000,E1 90.745} C_DIS
LIN {X 0.171,Y -576.948,Z 1401.304,A 0.000,B 0.000,C 90.000,E1 90.630} C_DIS
LIN {X -0.102,Y -573.983,Z 1401.302,A 0.000,B 0.000,C 90.000,E1 90.344} C_DIS
LIN {X -0.144,Y -573.971,Z 1401.302,A 0.000,B 0.000,C 90.000,E1 90.344} C_DIS
LIN {X -0.037,Y -573.378,Z 1401.300,A 0.000,B 0.000,C 90.000,E1 90.057} C_DIS
LIN {X -0.109,Y -573.316,Z 1401.298,A 0.000,B 0.000,C 90.000,E1 89.656} C_DIS
LIN {X -0.234,Y -574.916,Z 1401.287,A 0.000,B 0.000,C 90.000,E1 87.764} C_DIS
LIN {X 0.098,Y -576.318,Z 1401.278,A 0.000,B 0.000,C 90.000,E1 86.102} C_DIS
LIN {X 0.112,Y -578.231,Z 1401.268,A 0.000,B 0.000,C 90.000,E1 84.204} C_DIS
LIN {X 0.240,Y -580.376,Z 1401.257,A 0.000,B 0.000,C 90.000,E1 82.299} C_DIS
LIN {X 0.270,Y -582.263,Z 1401.248,A 0.000,B 0.000,C 90.000,E1 80.679} C_DIS
LIN {X -0.045,Y -583.481,Z 1401.242,A 0.000,B 0.000,C 90.000,E1 79.634} C_DIS
LIN {X -0.234,Y -584.686,Z 1401.236,A 0.000,B 0.000,C 90.000,E1 78.578} C_DIS
LIN {X -0.153,Y -585.924,Z 1401.229,A 0.000,B 0.000,C 90.000,E1 77.229} C_DIS
LIN {X 0.016,Y -587.434,Z 1401.219,A 0.000,B 0.000,C 90.000,E1 75.338} C_DIS
LIN {X 0.281,Y -588.304,Z 1401.211,A 0.000,B 0.000,C 90.000,E1 73.976} C_DIS
LIN {X -0.159,Y -589.180,Z 1401.202,A 0.000,B 0.000,C 90.000,E1 72.417} C_DIS
LIN {X -0.268,Y -589.930,Z 1401.195,A 0.000,B 0.000,C 90.000,E1 71.094} C_DIS
LIN {X 0.262,Y -590.837,Z 1401.186,A 0.000,B 0.000,C 90.000,E1 69.444} C_DIS
LIN {X -0.072,Y -591.956,Z 1401.176,A 0.000,B 0.000,C 90.000,E1 67.614} C_DIS
LIN {X 0.060,Y -593.227,Z 1401.165,A 0.000,B 0.000,C 90.000,E1 65.741} C_DIS
LIN {X -0.158,Y -594.918,Z 1401.154,A 0.000,B 0.000,C 90.000,E1 63.640} C_DIS
LIN {X 0.015,Y -595.755,Z 1401.148,A 0.000,B 0.000,C 90.000,E1 62.564} C_DIS
LIN {X 0.058,Y -597.038,Z 1401.139,A 0.000,B 0.000,C 90.000,E1 60.973} C_DIS
LIN {X -0.069,Y -598.256,Z 1401.131,A 0.000,B 0.000,C 90.000,E1 59.665} C_DIS
LIN {X 0.035,Y -599.737,Z 1401.123,A 0.000,B 0.000,C 90.000,E1 58.074} C_DIS
LIN {X -0.026,Y -601.205,Z 1401.114,A 0.000,B 0.000,C 90.000,E1 56.501} C_DIS
LIN {X -0.306,Y -602.842,Z 1401.104,A 0.000,B 0.000,C 90.000,E1 54.689} C_DIS
LIN {X 0.028,Y -604.240,Z 1401.095,A 0.000,B 0.000,C 90.000,E1 53.084} C_DIS
LIN {X 0.000,Y -605.210,Z 1401.088,A 0.000,B 0.000,C 90.000,E1 51.778} C_DIS
LIN {X 0.105,Y -605.920,Z 1401.082,A 0.000,B 0.000,C 90.000,E1 50.723} C_DIS
LIN {X -0.100,Y -606.708,Z 1401.073,A 0.000,B 0.000,C 90.000,E1 49.175} C_DIS
LIN {X 0.050,Y -607.088,Z 1401.064,A 0.000,B 0.000,C 90.000,E1 47.595} C_DIS
LIN {X -0.009,Y -607.168,Z 1401.057,A 0.000,B 0.000,C 90.000,E1 46.296} C_DIS
LIN {X 0.097,Y -607.112,Z 1401.051,A 0.000,B 0.000,C 90.000,E1 45.243} C_DIS
LIN {X 0.203,Y -606.954,Z 1401.046,A 0.000,B 0.000,C 90.000,E1 44.190} C_DIS
LIN {X 0.360,Y -606.252,Z 1401.037,A 0.000,B 0.000,C 90.000,E1 42.609} C_DIS
LIN {X 0.031,Y -605.682,Z 1401.031,A 0.000,B 0.000,C 90.000,E1 41.595} C_DIS
LIN {X -0.056,Y -604.776,Z 1401.024,A 0.000,B 0.000,C 90.000,E1 40.297} C_DIS
LIN {X 0.253,Y -604.104,Z 1401.020,A 0.000,B 0.000,C 90.000,E1 39.483} C_DIS
LIN {X 0.217,Y -602.703,Z 1401.012,A 0.000,B 0.000,C 90.000,E1 38.177} C_DIS
LIN {X -0.342,Y -601.746,Z 1401.008,A 0.000,B 0.000,C 90.000,E1 37.443} C_DIS
LIN {X 0.065,Y -599.796,Z 1401.001,A 0.000,B 0.000,C 90.000,E1 36.091} C_DIS
LIN {X 0.195,Y -597.879,Z 1400.995,A 0.000,B 0.000,C 90.000,E1 35.025} C_DIS
LIN {X 0.061,Y -596.238,Z 1400.990,A 0.000,B 0.000,C 90.000,E1 34.246} C_DIS
LIN {X -0.312,Y -593.128,Z 1400.983,A 0.000,B 0.000,C 90.000,E1 32.959} C_DIS
LIN {X -0.003,Y -590.955,Z 1400.979,A 0.000,B 0.000,C 90.000,E1 32.133} C_DIS
LIN {X -0.033,Y -588.576,Z 1400.974,A 0.000,B 0.000,C 90.000,E1 31.337} C_DIS
LIN {X -0.081,Y -585.778,Z 1400.970,A 0.000,B 0.000,C 90.000,E1 30.541} C_DIS
LIN {X -0.031,Y -583.765,Z 1400.967,A 0.000,B 0.000,C 90.000,E1 30.001} C_DIS
LIN {X -0.132,Y -580.235,Z 1400.962,A 0.000,B 0.000,C 90.000,E1 29.205} C_DIS
LIN {X 0.379,Y -577.687,Z 1400.959,A 0.000,B 0.000,C 90.000,E1 28.615} C_DIS
LIN {X -0.067,Y -573.598,Z 1400.955,A 0.000,B 0.000,C 90.000,E1 27.847} C_DIS
LIN {X 0.221,Y -569.227,Z 1400.950,A 0.000,B 0.000,C 90.000,E1 27.001} C_DIS
LIN {X -0.215,Y -565.231,Z 1400.946,A 0.000,B 0.000,C 90.000,E1 26.360} C_DIS
LIN {X -0.172,Y -561.053,Z 1400.943,A 0.000,B 0.000,C 90.000,E1 25.668} C_DIS
LIN {X 0.070,Y -556.593,Z 1400.939,A 0.000,B 0.000,C 90.000,E1 24.951} C_DIS
LIN {X -0.081,Y -550.620,Z 1400.934,A 0.000,B 0.000,C 90.000,E1 24.131} C_DIS
LIN {X 0.072,Y -547.455,Z 1400.932,A 0.000,B 0.000,C 90.000,E1 23.695} C_DIS
LIN {X 0.111,Y -540.692,Z 1400.927,A 0.000,B 0.000,C 90.000,E1 22.845} C_DIS
LIN {X -0.067,Y -534.723,Z 1400.923,A 0.000,B 0.000,C 90.000,E1 22.153} C_DIS
LIN {X -0.023,Y -525.823,Z 1400.918,A 0.000,B 0.000,C 90.000,E1 21.153} C_DIS
LIN {X 0.272,Y -515.418,Z 1400.911,A 0.000,B 0.000,C 90.000,E1 19.993} C_DIS
LIN {X 0.163,Y -505.999,Z 1400.906,A 0.000,B 0.000,C 90.000,E1 19.033} C_DIS
LIN {X -0.135,Y -493.703,Z 1400.899,A 0.000,B 0.000,C 90.000,E1 17.819} C_DIS
LIN {X 0.059,Y -478.846,Z 1400.890,A 0.000,B 0.000,C 90.000,E1 16.260} C_DIS
LIN {X -0.007,Y -462.494,Z 1400.881,A 0.000,B 0.000,C 90.000,E1 14.537} C_DIS
LIN {X -0.125,Y -450.307,Z 1400.874,A 0.000,B 0.000,C 90.000,E1 13.244} C_DIS
LIN {X -0.049,Y -439.213,Z 1400.867,A 0.000,B 0.000,C 90.000,E1 12.007} C_DIS
LIN {X 0.092,Y -429.559,Z 1400.861,A 0.000,B 0.000,C 90.000,E1 10.894} C_DIS
LIN {X 0.043,Y -411.956,Z 1400.849,A 0.000,B 0.000,C 90.000,E1 8.746} C_DIS
LIN {X -0.148,Y -402.606,Z 1400.842,A 0.000,B 0.000,C 90.000,E1 7.587} C_DIS
LIN {X -0.169,Y -393.125,Z 1400.835,A 0.000,B 0.000,C 90.000,E1 6.372} C_DIS
LIN {X -0.011,Y -389.180,Z 1400.832,A 0.000,B 0.000,C 90.000,E1 5.739} C_DIS
LIN {X 0.174,Y -388.268,Z 1400.830,A 0.000,B 0.000,C 90.000,E1 5.454} C_DIS
LIN {X 0.135,Y -388.248,Z 1400.830,A 0.000,B 0.000,C 90.000,E1 5.454} C_DIS
LIN {X 0.076,Y -388.464,Z 1400.830,A 0.000,B 0.000,C 90.000,E1 5.334} C_DIS
LIN {X 0.039,Y -388.487,Z 1400.830,A 0.000,B 0.000,C 90.000,E1 5.334} C_DIS
LIN {X 0.151,Y -393.359,Z 1400.827,A 0.000,B 0.000,C 90.000,E1 4.759} C_DIS
LIN {X 0.023,Y -399.871,Z 1400.823,A 0.000,B 0.000,C 90.000,E1 4.188} C_DIS
LIN {X -0.182,Y -404.372,Z 1400.821,A 0.000,B 0.000,C 90.000,E1 3.784} C_DIS
LIN {X 0.006,Y -405.764,Z 1400.820,A 0.000,B 0.000,C 90.000,E1 3.612} C_DIS
LIN {X -0.192,Y -409.731,Z 1400.817,A 0.000,B 0.000,C 90.000,E1 3.151} C_DIS
LIN {X -0.143,Y -412.579,Z 1400.816,A 0.000,B 0.000,C 90.000,E1 2.808} C_DIS
LIN {X -0.133,Y -418.687,Z 1400.811,A 0.000,B 0.000,C 90.000,E1 1.949} C_DIS
LIN {X -0.004,Y -426.217,Z 1400.804,A 0.000,B 0.000,C 90.000,E1 0.745} C_DIS
LIN {X 0.000,Y -430.772,Z 1400.800,A 0.000,B 0.000,C 90.000,E1 360.000} C_DIS
LIN {X -0.058,Y -436.762,Z 1400.794,A 0.000,B 0.000,C 90.000,E1 358.969} C_DIS
LIN {X 0.145,Y -440.245,Z 1400.791,A 0.000,B 0.000,C 90.000,E1 358.282} C_DIS
LIN {X -0.109,Y -442.421,Z 1400.788,A 0.000,B 0.000,C 90.000,E1 357.822} C_DIS
LIN {X 0.012,Y -443.665,Z 1400.786,A 0.000,B 0.000,C 90.000,E1 357.478} C_DIS
LIN {X 0.139,Y -444.573,Z 1400.784,A 0.000,B 0.000,C 90.000,E1 357.135} C_DIS
LIN {X -0.153,Y -444.987,Z 1400.782,A 0.000,B 0.000,C 90.000,E1 356.846} C_DIS
LIN {X -0.021,Y -444.367,Z 1400.781,A 0.000,B 0.000,C 90.000,E1 356.502} C_DIS
LIN {X -0.014,Y -443.920,Z 1400.780,A 0.000,B 0.000,C 90.000,E1 356.445} C_DIS
LIN {X 0.036,Y -443.089,Z 1400.780,A 0.000,B 0.000,C 90.000,E1 356.388} C_DIS
LIN {X 0.039,Y -430.428,Z 1400.779,A 0.000,B 0.000,C 90.000,E1 356.274} C_DIS
LIN {X 0.133,Y -373.081,Z 1400.776,A 0.000,B 0.000,C 90.000,E1 355.698} C_DIS
LIN {X -0.141,Y -359.592,Z 1400.775,A 0.000,B 0.000,C 90.000,E1 355.584} C_DIS
LIN {X -0.163,Y -359.427,Z 1400.775,A 0.000,B 0.000,C 90.000,E1 355.584} C_DIS
LIN {X 0.177,Y -359.434,Z 1400.769,A 0.000,B 0.000,C 90.000,E1 354.375} C_DIS
LIN {X -0.081,Y -359.586,Z 1400.725,A 0.000,B 0.000,C 90.000,E1 346.520} C_DIS
LIN {X -0.169,Y -361.898,Z 1400.683,A 0.000,B 0.000,C 90.000,E1 339.028} C_DIS
LIN {X 0.076,Y -365.750,Z 1400.644,A 0.000,B 0.000,C 90.000,E1 331.897} C_DIS
LIN {X 0.156,Y -366.110,Z 1400.642,A 0.000,B 0.000,C 90.000,E1 331.513} C_DIS
LIN {X -0.123,Y -370.671,Z 1400.607,A 0.000,B 0.000,C 90.000,E1 325.261} C_DIS
LIN {X 0.150,Y -371.510,Z 1400.603,A 0.000,B 0.000,C 90.000,E1 324.482} C_DIS
LIN {X -0.088,Y -372.046,Z 1400.599,A 0.000,B 0.000,C 90.000,E1 323.783} C_DIS
LIN {X -0.049,Y -378.006,Z 1400.564,A 0.000,B 0.000,C 90.000,E1 317.553} C_DIS
LIN {X 0.003,Y -379.688,Z 1400.552,A 0.000,B 0.000,C 90.000,E1 315.364} C_DIS
LIN {X 0.011,Y -384.614,Z 1400.528,A 0.000,B 0.000,C 90.000,E1 311.024} C_DIS
LIN {X 0.063,Y -385.220,Z 1400.524,A 0.000,B 0.000,C 90.000,E1 310.297} C_DIS
LIN {X -0.221,Y -391.274,Z 1400.492,A 0.000,B 0.000,C 90.000,E1 304.612} C_DIS
LIN {X -0.067,Y -396.986,Z 1400.459,A 0.000,B 0.000,C 90.000,E1 298.565} C_DIS
LIN {X -0.116,Y -401.350,Z 1400.427,A 0.000,B 0.000,C 90.000,E1 292.950} C_DIS
LIN {X -0.036,Y -401.658,Z 1400.426,A 0.000,B 0.000,C 90.000,E1 292.589} C_DIS
LIN {X 0.116,Y -404.748,Z 1400.395,A 0.000,B 0.000,C 90.000,E1 286.985} C_DIS
LIN {X 0.130,Y -406.156,Z 1400.364,A 0.000,B 0.000,C 90.000,E1 281.422} C_DIS
LIN {X -0.170,Y -405.676,Z 1400.333,A 0.000,B 0.000,C 90.000,E1 275.910} C_DIS
LIN {X -0.098,Y -403.565,Z 1400.306,A 0.000,B 0.000,C 90.000,E1 271.031} C_DIS
LIN {X -0.163,Y -403.173,Z 1400.302,A 0.000,B 0.000,C 90.000,E1 270.344} C_DIS
LIN {X 0.070,Y -399.063,Z 1400.273,A 0.000,B 0.000,C 90.000,E1 265.065} C_DIS
LIN {X 0.011,Y -398.765,Z 1400.271,A 0.000,B 0.000,C 90.000,E1 264.723} C_DIS
LIN {X -0.099,Y -393.286,Z 1400.243,A 0.000,B 0.000,C 90.000,E1 259.803} C_DIS
LIN {X -0.177,Y -392.659,Z 1400.239,A 0.000,B 0.000,C 90.000,E1 259.106} C_DIS
LIN {X -0.006,Y -386.239,Z 1400.214,A 0.000,B 0.000,C 90.000,E1 254.448} C_DIS
LIN {X -0.041,Y -385.141,Z 1400.208,A 0.000,B 0.000,C 90.000,E1 253.378} C_DIS
LIN {X 0.067,Y -377.806,Z 1400.182,A 0.000,B 0.000,C 90.000,E1 248.666} C_DIS
LIN {X -0.061,Y -376.074,Z 1400.173,A 0.000,B 0.000,C 90.000,E1 247.230} C_DIS
LIN {X -0.003,Y -368.743,Z 1400.149,A 0.000,B 0.000,C 90.000,E1 242.820} C_DIS
LIN {X -0.018,Y -366.390,Z 1400.139,A 0.000,B 0.000,C 90.000,E1 240.973} C_DIS
LIN {X 0.147,Y -365.088,Z 1400.135,A 0.000,B 0.000,C 90.000,E1 240.205} C_DIS
LIN {X -0.104,Y -358.493,Z 1400.112,A 0.000,B 0.000,C 90.000,E1 236.135} C_DIS
LIN {X -0.045,Y -356.170,Z 1400.101,A 0.000,B 0.000,C 90.000,E1 234.242} C_DIS
LIN {X -0.104,Y -354.919,Z 1400.097,A 0.000,B 0.000,C 90.000,E1 233.497} C_DIS
LIN {X -0.120,Y -348.151,Z 1400.072,A 0.000,B 0.000,C 90.000,E1 228.933} C_DIS
LIN {X 0.050,Y -346.048,Z 1400.061,A 0.000,B 0.000,C 90.000,E1 226.986} C_DIS
LIN {X 0.022,Y -339.247,Z 1400.033,A 0.000,B 0.000,C 90.000,E1 221.962} C_DIS
LIN {X -0.114,Y -337.051,Z 1400.020,A 0.000,B 0.000,C 90.000,E1 219.644} C_DIS
LIN {X 0.219,Y -336.658,Z 1400.018,A 0.000,B 0.000,C 90.000,E1 219.197} C_DIS
LIN {X 0.115,Y -330.751,Z 1399.987,A 0.000,B 0.000,C 90.000,E1 213.706} C_DIS
LIN {X 0.067,Y -329.193,Z 1399.974,A 0.000,B 0.000,C 90.000,E1 211.337} C_DIS
LIN {X 0.101,Y -324.429,Z 1399.939,A 0.000,B 0.000,C 90.000,E1 204.951} C_DIS
LIN {X 0.085,Y -323.758,Z 1399.928,A 0.000,B 0.000,C 90.000,E1 202.950} C_DIS
LIN {X -0.124,Y -321.139,Z 1399.881,A 0.000,B 0.000,C 90.000,E1 194.537} C_DIS
LIN {X 0.075,Y -321.598,Z 1399.831,A 0.000,B 0.000,C 90.000,E1 185.625} C_DIS
LIN {X -0.116,Y -321.598,Z 1399.831,A 0.000,B 0.000,C 90.000,E1 185.511} C_DIS
LIN {X -0.142,Y -321.645,Z 1399.831,A 0.000,B 0.000,C 90.000,E1 185.511} C_DIS
LIN {X 0.069,Y -366.482,Z 1399.827,A 0.000,B 0.000,C 90.000,E1 184.821} C_DIS
LIN {X 0.158,Y -410.631,Z 1399.824,A 0.000,B 0.000,C 90.000,E1 184.302} C_DIS
LIN {X -0.191,Y -414.059,Z 1399.824,A 0.000,B 0.000,C 90.000,E1 184.302} C_DIS
LIN {X -0.204,Y -414.833,Z 1399.823,A 0.000,B 0.000,C 90.000,E1 184.245} C_DIS
LIN {X 0.114,Y -415.898,Z 1399.822,A 0.000,B 0.000,C 90.000,E1 183.955} C_DIS
LIN {X 0.121,Y -416.080,Z 1399.820,A 0.000,B 0.000,C 90.000,E1 183.612} C_DIS
LIN {X 0.134,Y -415.759,Z 1399.818,A 0.000,B 0.000,C 90.000,E1 183.269} C_DIS
LIN {X 0.171,Y -415.198,Z 1399.816,A 0.000,B 0.000,C 90.000,E1 182.922} C_DIS
LIN {X -0.207,Y -412.972,Z 1399.811,A 0.000,B 0.000,C 90.000,E1 181.949} C_DIS
LIN {X -0.183,Y -411.304,Z 1399.807,A 0.000,B 0.000,C 90.000,E1 181.260} C_DIS
LIN {X -0.188,Y -408.294,Z 1399.801,A 0.000,B 0.000,C 90.000,E1 180.229} C_DIS
LIN {X 0.196,Y -406.017,Z 1399.797,A 0.000,B 0.000,C 90.000,E1 179.484} C_DIS
LIN {X 0.121,Y -402.193,Z 1399.792,A 0.000,B 0.000,C 90.000,E1 178.453} C_DIS
LIN {X 0.031,Y -398.482,Z 1399.787,A 0.000,B 0.000,C 90.000,E1 177.593} C_DIS
LIN {X -0.123,Y -393.052,Z 1399.781,A 0.000,B 0.000,C 90.000,E1 176.560} C_DIS
LIN {X 0.044,Y -386.807,Z 1399.775,A 0.000,B 0.000,C 90.000,E1 175.469} C_DIS
LIN {X -0.138,Y -375.388,Z 1399.764,A 0.000,B 0.000,C 90.000,E1 173.514} C_DIS
LIN {X -0.113,Y -369.616,Z 1399.758,A 0.000,B 0.000,C 90.000,E1 172.413} C_DIS
LIN {X 0.060,Y -362.514,Z 1399.750,A 0.000,B 0.000,C 90.000,E1 170.905} C_DIS
LIN {X -0.094,Y -360.915,Z 1399.748,A 0.000,B 0.000,C 90.000,E1 170.557} C_DIS
LIN {X -0.182,Y -357.816,Z 1399.742,A 0.000,B 0.000,C 90.000,E1 169.634} C_DIS
LIN {X -0.142,Y -357.276,Z 1399.740,A 0.000,B 0.000,C 90.000,E1 169.275} C_DIS
LIN {X 0.180,Y -357.289,Z 1399.740,A 0.000,B 0.000,C 90.000,E1 169.218} C_DIS
LIN {X 0.111,Y -357.758,Z 1399.740,A 0.000,B 0.000,C 90.000,E1 169.106} C_DIS
LIN {X -0.141,Y -358.949,Z 1399.737,A 0.000,B 0.000,C 90.000,E1 168.701} C_DIS
LIN {X -0.159,Y -358.964,Z 1399.737,A 0.000,B 0.000,C 90.000,E1 168.701} C_DIS
LIN {X 0.055,Y -362.016,Z 1399.734,A 0.000,B 0.000,C 90.000,E1 168.173} C_DIS
LIN {X 0.124,Y -368.929,Z 1399.729,A 0.000,B 0.000,C 90.000,E1 167.229} C_DIS
LIN {X -0.164,Y -376.085,Z 1399.724,A 0.000,B 0.000,C 90.000,E1 166.408} C_DIS
LIN {X -0.135,Y -389.581,Z 1399.716,A 0.000,B 0.000,C 90.000,E1 164.936} C_DIS
LIN {X 0.083,Y -400.030,Z 1399.710,A 0.000,B 0.000,C 90.000,E1 163.866} C_DIS
LIN {X 0.203,Y -414.045,Z 1399.703,A 0.000,B 0.000,C 90.000,E1 162.598} C_DIS
LIN {X -0.178,Y -431.412,Z 1399.696,A 0.000,B 0.000,C 90.000,E1 161.221} C_DIS
LIN {X 0.046,Y -442.440,Z 1399.691,A 0.000,B 0.000,C 90.000,E1 160.315} C_DIS
LIN {X 0.025,Y -453.365,Z 1399.686,A 0.000,B 0.000,C 90.000,E1 159.444} C_DIS
LIN {X -0.198,Y -464.030,Z 1399.681,A 0.000,B 0.000,C 90.000,E1 158.592} C_DIS
LIN {X 0.086,Y -471.568,Z 1399.677,A 0.000,B 0.000,C 90.000,E1 157.922} C_DIS
LIN {X -0.043,Y -478.822,Z 1399.674,A 0.000,B 0.000,C 90.000,E1 157.283} C_DIS
LIN {X -0.217,Y -490.338,Z 1399.668,A 0.000,B 0.000,C 90.000,E1 156.230} C_DIS
LIN {X 0.009,Y -495.908,Z 1399.665,A 0.000,B 0.000,C 90.000,E1 155.665} C_DIS
LIN {X 0.216,Y -500.031,Z 1399.663,A 0.000,B 0.000,C 90.000,E1 155.229} C_DIS
LIN {X -0.203,Y -505.322,Z 1399.659,A 0.000,B 0.000,C 90.000,E1 154.717} C_DIS
LIN {X -0.006,Y -511.780,Z 1399.655,A 0.000,B 0.000,C 90.000,E1 153.973} C_DIS
LIN {X 0.191,Y -515.507,Z 1399.653,A 0.000,B 0.000,C 90.000,E1 153.512} C_DIS
LIN {X 0.037,Y -521.329,Z 1399.649,A 0.000,B 0.000,C 90.000,E1 152.794} C_DIS
LIN {X 0.014,Y -524.548,Z 1399.646,A 0.000,B 0.000,C 90.000,E1 152.359} C_DIS
LIN {X 0.251,Y -527.556,Z 1399.644,A 0.000,B 0.000,C 90.000,E1 151.897} C_DIS
LIN {X -0.210,Y -530.360,Z 1399.642,A 0.000,B 0.000,C 90.000,E1 151.513} C_DIS
LIN {X -0.086,Y -533.690,Z 1399.638,A 0.000,B 0.000,C 90.000,E1 150.923} C_DIS
LIN {X -0.078,Y -537.169,Z 1399.635,A 0.000,B 0.000,C 90.000,E1 150.205} C_DIS
LIN {X 0.097,Y -539.583,Z 1399.631,A 0.000,B 0.000,C 90.000,E1 149.616} C_DIS
LIN {X -0.170,Y -542.698,Z 1399.627,A 0.000,B 0.000,C 90.000,E1 148.791} C_DIS
LIN {X 0.041,Y -544.572,Z 1399.623,A 0.000,B 0.000,C 90.000,E1 148.201} C_DIS
LIN {X -0.200,Y -546.268,Z 1399.620,A 0.000,B 0.000,C 90.000,E1 147.661} C_DIS
LIN {X 0.068,Y -548.399,Z 1399.616,A 0.000,B 0.000,C 90.000,E1 146.786} C_DIS
LIN {X -0.102,Y -550.212,Z 1399.611,A 0.000,B 0.000,C 90.000,E1 145.960} C_DIS
LIN {X 0.060,Y -551.739,Z 1399.606,A 0.000,B 0.000,C 90.000,E1 145.102} C_DIS
LIN {X -0.137,Y -552.578,Z 1399.603,A 0.000,B 0.000,C 90.000,E1 144.562} C_DIS
LIN {X 0.057,Y -553.504,Z 1399.598,A 0.000,B 0.000,C 90.000,E1 143.703} C_DIS
LIN {X -0.031,Y -554.857,Z 1399.591,A 0.000,B 0.000,C 90.000,E1 142.316} C_DIS
LIN {X -0.014,Y -556.282,Z 1399.581,A 0.000,B 0.000,C 90.000,E1 140.642} C_DIS
LIN {X -0.137,Y -557.170,Z 1399.575,A 0.000,B 0.000,C 90.000,E1 139.542} C_DIS
LIN {X -0.161,Y -558.071,Z 1399.566,A 0.000,B 0.000,C 90.000,E1 137.877} C_DIS
LIN {X 0.132,Y -558.627,Z 1399.558,A 0.000,B 0.000,C 90.000,E1 136.458} C_DIS
LIN {X 0.038,Y -559.182,Z 1399.551,A 0.000,B 0.000,C 90.000,E1 135.081} C_DIS
LIN {X 0.287,Y -559.496,Z 1399.544,A 0.000,B 0.000,C 90.000,E1 133.947} C_DIS
LIN {X -0.102,Y -559.890,Z 1399.535,A 0.000,B 0.000,C 90.000,E1 132.324} C_DIS
LIN {X -0.231,Y -560.011,Z 1399.529,A 0.000,B 0.000,C 90.000,E1 131.229} C_DIS
LIN {X -0.192,Y -560.260,Z 1399.520,A 0.000,B 0.000,C 90.000,E1 129.564} C_DIS
LIN {X -0.070,Y -560.665,Z 1399.510,A 0.000,B 0.000,C 90.000,E1 127.890} C_DIS
LIN {X 0.151,Y -560.758,Z 1399.500,A 0.000,B 0.000,C 90.000,E1 125.931} C_DIS
LIN {X 0.264,Y -561.496,Z 1399.487,A 0.000,B 0.000,C 90.000,E1 123.706} C_DIS
LIN {X 0.248,Y -561.875,Z 1399.485,A 0.000,B 0.000,C 90.000,E1 123.293} C_DIS
LIN {X -0.007,Y -563.259,Z 1399.482,A 0.000,B 0.000,C 90.000,E1 122.704} C_DIS
LIN {X 0.024,Y -564.737,Z 1399.481,A 0.000,B 0.000,C 90.000,E1 122.546} C_DIS
LIN {X 0.124,Y -565.820,Z 1399.480,A 0.000,B 0.000,C 90.000,E1 122.467} C_DIS
LIN {X -0.079,Y -567.914,Z 1399.480,A 0.000,B 0.000,C 90.000,E1 122.418} C_DIS
LIN {X 0.140,Y -573.156,Z 1399.479,A 0.000,B 0.000,C 90.000,E1 122.260} C_DIS
LIN {X 0.301,Y -578.283,Z 1399.479,A 0.000,B 0.000,C 90.000,E1 122.133} C_DIS
LIN {X -0.036,Y -581.889,Z 1399.478,A 0.000,B 0.000,C 90.000,E1 122.084} C_DIS
LIN {X 0.124,Y -584.004,Z 1399.478,A 0.000,B 0.000,C 90.000,E1 122.005} C_DIS
LIN {X -0.263,Y -589.762,Z 1399.477,A 0.000,B 0.000,C 90.000,E1 121.799} C_DIS
LIN {X -0.223,Y -595.358,Z 1399.475,A 0.000,B 0.000,C 90.000,E1 121.465} C_DIS
LIN {X -0.113,Y -600.988,Z 1399.473,A 0.000,B 0.000,C 90.000,E1 121.052} C_DIS
LIN {X -0.036,Y -605.161,Z 1399.471,A 0.000,B 0.000,C 90.000,E1 120.718} C_DIS
LIN {X -0.195,Y -610.251,Z 1399.468,A 0.000,B 0.000,C 90.000,E1 120.256} C_DIS
LIN {X -0.092,Y -613.917,Z 1399.466,A 0.000,B 0.000,C 90.000,E1 119.873} C_DIS
LIN {X 0.204,Y -619.186,Z 1399.462,A 0.000,B 0.000,C 90.000,E1 119.205} C_DIS
LIN {X 0.183,Y -622.990,Z 1399.460,A 0.000,B 0.000,C 90.000,E1 118.693} C_DIS
LIN {X -0.361,Y -626.229,Z 1399.457,A 0.000,B 0.000,C 90.000,E1 118.231} C_DIS
LIN {X -0.333,Y -628.938,Z 1399.454,A 0.000,B 0.000,C 90.000,E1 117.719} C_DIS
LIN {X -0.008,Y -630.582,Z 1399.452,A 0.000,B 0.000,C 90.000,E1 117.308} C_DIS
LIN {X 0.016,Y -631.559,Z 1399.450,A 0.000,B 0.000,C 90.000,E1 117.052} C_DIS
LIN {X 0.046,Y -632.258,Z 1399.449,A 0.000,B 0.000,C 90.000,E1 116.796} C_DIS
LIN {X 0.077,Y -632.722,Z 1399.448,A 0.000,B 0.000,C 90.000,E1 116.539} C_DIS
LIN {X 0.112,Y -633.002,Z 1399.446,A 0.000,B 0.000,C 90.000,E1 116.283} C_DIS
LIN {X -0.052,Y -633.081,Z 1399.442,A 0.000,B 0.000,C 90.000,E1 115.540} C_DIS
LIN {X 0.025,Y -632.045,Z 1399.439,A 0.000,B 0.000,C 90.000,E1 115.027} C_DIS
LIN {X 0.061,Y -630.959,Z 1399.438,A 0.000,B 0.000,C 90.000,E1 114.771} C_DIS
LIN {X 0.106,Y -628.767,Z 1399.436,A 0.000,B 0.000,C 90.000,E1 114.387} C_DIS
LIN {X 0.120,Y -627.822,Z 1399.435,A 0.000,B 0.000,C 90.000,E1 114.259} C_DIS
LIN {X 0.129,Y -622.237,Z 1399.432,A 0.000,B 0.000,C 90.000,E1 113.770} C_DIS
LIN {X 0.107,Y -615.053,Z 1399.430,A 0.000,B 0.000,C 90.000,E1 113.387} C_DIS
LIN {X -0.245,Y -613.261,Z 1399.430,A 0.000,B 0.000,C 90.000,E1 113.334} C_DIS
LIN {X 0.258,Y -607.526,Z 1399.428,A 0.000,B 0.000,C 90.000,E1 113.078} C_DIS
LIN {X 0.370,Y -604.830,Z 1399.428,A 0.000,B 0.000,C 90.000,E1 112.950} C_DIS
LIN {X 0.168,Y -596.791,Z 1399.426,A 0.000,B 0.000,C 90.000,E1 112.717} C_DIS
LIN {X -0.025,Y -594.818,Z 1399.426,A 0.000,B 0.000,C 90.000,E1 112.642} C_DIS
LIN {X -0.067,Y -594.858,Z 1399.426,A 0.000,B 0.000,C 90.000,E1 112.642} C_DIS
LIN {X 0.154,Y -606.520,Z 1399.421,A 0.000,B 0.000,C 90.000,E1 111.770} C_DIS
LIN {X 0.056,Y -613.324,Z 1399.418,A 0.000,B 0.000,C 90.000,E1 111.227} C_DIS
LIN {X -0.326,Y -617.270,Z 1399.416,A 0.000,B 0.000,C 90.000,E1 110.918} C_DIS
LIN {X -0.150,Y -623.417,Z 1399.413,A 0.000,B 0.000,C 90.000,E1 110.301} C_DIS
LIN {X -0.283,Y -626.977,Z 1399.411,A 0.000,B 0.000,C 90.000,E1 109.939} C_DIS
LIN {X 0.122,Y -632.183,Z 1399.407,A 0.000,B 0.000,C 90.000,E1 109.268} C_DIS
LIN {X -0.037,Y -635.922,Z 1399.404,A 0.000,B 0.000,C 90.000,E1 108.779} C_DIS
LIN {X 0.232,Y -640.856,Z 1399.400,A 0.000,B 0.000,C 90.000,E1 108.000} C_DIS
LIN {X -0.079,Y -644.316,Z 1399.397,A 0.000,B 0.000,C 90.000,E1 107.402} C_DIS
LIN {X -0.195,Y -646.480,Z 1399.394,A 0.000,B 0.000,C 90.000,E1 106.913} C_DIS
LIN {X 0.276,Y -647.499,Z 1399.393,A 0.000,B 0.000,C 90.000,E1 106.622} C_DIS
LIN {X 0.174,Y -649.004,Z 1399.390,A 0.000,B 0.000,C 90.000,E1 106.134} C_DIS
LIN {X 0.036,Y -649.640,Z 1399.388,A 0.000,B 0.000,C 90.000,E1 105.898} C_DIS
LIN {X -0.233,Y -650.627,Z 1399.386,A 0.000,B 0.000,C 90.000,E1 105.426} C_DIS
LIN {X 0.010,Y -651.722,Z 1399.381,A 0.000,B 0.000,C 90.000,E1 104.662} C_DIS
LIN {X -0.204,Y -652.626,Z 1399.377,A 0.000,B 0.000,C 90.000,E1 103.939} C_DIS
LIN {X 0.059,Y -653.248,Z 1399.373,A 0.000,B 0.000,C 90.000,E1 103.175} C_DIS
LIN {X -0.186,Y -653.337,Z 1399.370,A 0.000,B 0.000,C 90.000,E1 102.703} C_DIS
LIN {X 0.330,Y -653.353,Z 1399.369,A 0.000,B 0.000,C 90.000,E1 102.411} C_DIS
LIN {X -0.173,Y -652.954,Z 1399.365,A 0.000,B 0.000,C 90.000,E1 101.715} C_DIS
LIN {X 0.219,Y -652.505,Z 1399.362,A 0.000,B 0.000,C 90.000,E1 101.186} C_DIS
LIN {X -0.282,Y -651.483,Z 1399.358,A 0.000,B 0.000,C 90.000,E1 100.489} C_DIS
LIN {X 0.229,Y -651.090,Z 1399.357,A 0.000,B 0.000,C 90.000,E1 100.197} C_DIS
LIN {X -0.284,Y -649.291,Z 1399.353,A 0.000,B 0.000,C 90.000,E1 99.500} C_DIS
LIN {X 0.075,Y -647.885,Z 1399.350,A 0.000,B 0.000,C 90.000,E1 98.973} C_DIS
LIN {X -0.318,Y -646.260,Z 1399.347,A 0.000,B 0.000,C 90.000,E1 98.511} C_DIS
LIN {X -0.078,Y -644.433,Z 1399.344,A 0.000,B 0.000,C 90.000,E1 97.992} C_DIS
LIN {X -0.017,Y -641.217,Z 1399.340,A 0.000,B 0.000,C 90.000,E1 97.239} C_DIS
LIN {X 0.317,Y -639.470,Z 1399.338,A 0.000,B 0.000,C 90.000,E1 96.834} C_DIS
LIN {X 0.244,Y -635.429,Z 1399.334,A 0.000,B 0.000,C 90.000,E1 96.087} C_DIS
LIN {X 0.196,Y -631.086,Z 1399.330,A 0.000,B 0.000,C 90.000,E1 95.334} C_DIS
LIN {X 0.184,Y -627.118,Z 1399.326,A 0.000,B 0.000,C 90.000,E1 94.702} C_DIS
LIN {X 0.091,Y -622.438,Z 1399.323,A 0.000,B 0.000,C 90.000,E1 94.073} C_DIS
LIN {X 0.160,Y -617.899,Z 1399.320,A 0.000,B 0.000,C 90.000,E1 93.555} C_DIS
LIN {X -0.205,Y -610.201,Z 1399.316,A 0.000,B 0.000,C 90.000,E1 92.865} C_DIS
LIN {X 0.148,Y -601.983,Z 1399.312,A 0.000,B 0.000,C 90.000,E1 92.121} C_DIS
LIN {X 0.113,Y -596.317,Z 1399.309,A 0.000,B 0.000,C 90.000,E1 91.661} C_DIS
LIN {X -0.249,Y -590.129,Z 1399.307,A 0.000,B 0.000,C 90.000,E1 91.260} C_DIS
LIN {X -0.270,Y -584.876,Z 1399.305,A 0.000,B 0.000,C 90.000,E1 90.974} C_DIS
LIN {X 0.032,Y -577.763,Z 1399.303,A 0.000,B 0.000,C 90.000,E1 90.573} C_DIS
LIN {X -0.125,Y -575.266,Z 1399.302,A 0.000,B 0.000,C 90.000,E1 90.344} C_DIS
LIN {X 0.133,Y -574.172,Z 1399.301,A 0.000,B 0.000,C 90.000,E1 90.229} C_DIS
LIN {X 0.091,Y -574.130,Z 1399.301,A 0.000,B 0.000,C 90.000,E1 90.229} C_DIS
LIN {X -0.187,Y -573.471,Z 1399.300,A 0.000,B 0.000,C 90.000,E1 89.943} C_DIS
LIN {X 0.135,Y -573.399,Z 1399.297,A 0.000,B 0.000,C 90.000,E1 89.484} C_DIS
LIN {X 0.012,Y -575.008,Z 1399.287,A 0.000,B 0.000,C 90.000,E1 87.593} C_DIS
LIN {X -0.232,Y -576.414,Z 1399.278,A 0.000,B 0.000,C 90.000,E1 85.988} C_DIS
LIN {X -0.219,Y -578.360,Z 1399.267,A 0.000,B 0.000,C 90.000,E1 84.090} C_DIS
LIN {X -0.236,Y -580.203,Z 1399.258,A 0.000,B 0.000,C 90.000,E1 82.470} C_DIS
LIN {X -0.203,Y -582.106,Z 1399.249,A 0.000,B 0.000,C 90.000,E1 80.849} C_DIS
LIN {X 0.058,Y -583.344,Z 1399.243,A 0.000,B 0.000,C 90.000,E1 79.746} C_DIS
LIN {X -0.003,Y -584.816,Z 1399.236,A 0.000,B 0.000,C 90.000,E1 78.409} C_DIS
LIN {X 0.072,Y -586.031,Z 1399.228,A 0.000,B 0.000,C 90.000,E1 77.061} C_DIS
LIN {X 0.305,Y -587.083,Z 1399.221,A 0.000,B 0.000,C 90.000,E1 75.700} C_DIS
LIN {X -0.089,Y -587.703,Z 1399.216,A 0.000,B 0.000,C 90.000,E1 74.936} C_DIS
LIN {X -0.232,Y -588.522,Z 1399.209,A 0.000,B 0.000,C 90.000,E1 73.614} C_DIS
LIN {X 0.134,Y -589.583,Z 1399.198,A 0.000,B 0.000,C 90.000,E1 71.710} C_DIS
LIN {X -0.232,Y -590.612,Z 1399.188,A 0.000,B 0.000,C 90.000,E1 69.880} C_DIS
LIN {X 0.087,Y -591.895,Z 1399.176,A 0.000,B 0.000,C 90.000,E1 67.720} C_DIS
LIN {X -0.011,Y -593.145,Z 1399.166,A 0.000,B 0.000,C 90.000,E1 65.869} C_DIS
LIN {X -0.232,Y -594.817,Z 1399.154,A 0.000,B 0.000,C 90.000,E1 63.768} C_DIS
LIN {X 0.126,Y -595.861,Z 1399.147,A 0.000,B 0.000,C 90.000,E1 62.410} C_DIS
LIN {X -0.019,Y -596.945,Z 1399.140,A 0.000,B 0.000,C 90.000,E1 61.101} C_DIS
LIN {X -0.146,Y -598.151,Z 1399.132,A 0.000,B 0.000,C 90.000,E1 59.793} C_DIS
LIN {X -0.041,Y -599.628,Z 1399.123,A 0.000,B 0.000,C 90.000,E1 58.201} C_DIS
LIN {X -0.101,Y -601.083,Z 1399.115,A 0.000,B 0.000,C 90.000,E1 56.628} C_DIS
LIN {X 0.297,Y -601.793,Z 1399.110,A 0.000,B 0.000,C 90.000,E1 55.801} C_DIS
LIN {X -0.221,Y -603.218,Z 1399.101,A 0.000,B 0.000,C 90.000,E1 54.276} C_DIS
LIN {X -0.001,Y -604.585,Z 1399.093,A 0.000,B 0.000,C 90.000,E1 52.683} C_DIS
LIN {X 0.253,Y -605.719,Z 1399.084,A 0.000,B 0.000,C 90.000,E1 51.090} C_DIS
LIN {X -0.014,Y -606.304,Z 1399.078,A 0.000,B 0.000,C 90.000,E1 50.070} C_DIS
LIN {X -0.151,Y -606.716,Z 1399.074,A 0.000,B 0.000,C 90.000,E1 49.299} C_DIS
LIN {X 0.048,Y -607.117,Z 1399.065,A 0.000,B 0.000,C 90.000,E1 47.715} C_DIS
LIN {X -0.041,Y -607.202,Z 1399.058,A 0.000,B 0.000,C 90.000,E1 46.419} C_DIS
LIN {X 0.078,Y -607.167,Z 1399.052,A 0.000,B 0.000,C 90.000,E1 45.364} C_DIS
LIN {X -0.247,Y -607.021,Z 1399.046,A 0.000,B 0.000,C 90.000,E1 44.352} C_DIS
LIN {X 0.105,Y -606.462,Z 1399.039,A 0.000,B 0.000,C 90.000,E1 43.014} C_DIS
LIN {X 0.040,Y -605.811,Z 1399.032,A 0.000,B 0.000,C 90.000,E1 41.714} C_DIS
LIN {X -0.033,Y -604.959,Z 1399.025,A 0.000,B 0.000,C 90.000,E1 40.415} C_DIS
LIN {X -0.181,Y -604.328,Z 1399.020,A 0.000,B 0.000,C 90.000,E1 39.644} C_DIS
LIN {X 0.049,Y -602.656,Z 1399.011,A 0.000,B 0.000,C 90.000,E1 38.051} C_DIS
LIN {X -0.142,Y -601.668,Z 1399.007,A 0.000,B 0.000,C 90.000,E1 37.282} C_DIS
LIN {X 0.012,Y -600.149,Z 1399.001,A 0.000,B 0.000,C 90.000,E1 36.217} C_DIS
LIN {X -0.096,Y -598.746,Z 1398.997,A 0.000,B 0.000,C 90.000,E1 35.438} C_DIS
LIN {X -0.324,Y -596.659,Z 1398.991,A 0.000,B 0.000,C 90.000,E1 34.405} C_DIS
LIN {X 0.139,Y -593.631,Z 1398.984,A 0.000,B 0.000,C 90.000,E1 33.038} C_DIS
LIN {X -0.046,Y -591.497,Z 1398.979,A 0.000,B 0.000,C 90.000,E1 32.260} C_DIS
LIN {X -0.185,Y -588.363,Z 1398.973,A 0.000,B 0.000,C 90.000,E1 31.209} C_DIS
LIN {X -0.061,Y -584.431,Z 1398.967,A 0.000,B 0.000,C 90.000,E1 30.129} C_DIS
LIN {X -0.155,Y -581.037,Z 1398.963,A 0.000,B 0.000,C 90.000,E1 29.333} C_DIS
LIN {X 0.288,Y -577.869,Z 1398.959,A 0.000,B 0.000,C 90.000,E1 28.615} C_DIS
LIN {X -0.233,Y -573.076,Z 1398.954,A 0.000,B 0.000,C 90.000,E1 27.719} C_DIS
LIN {X 0.134,Y -569.420,Z 1398.950,A 0.000,B 0.000,C 90.000,E1 27.001} C_DIS
LIN {X -0.298,Y -565.456,Z 1398.946,A 0.000,B 0.000,C 90.000,E1 26.360} C_DIS
LIN {X -0.109,Y -560.404,Z 1398.942,A 0.000,B 0.000,C 90.000,E1 25.515} C_DIS
LIN {X -0.113,Y -555.844,Z 1398.938,A 0.000,B 0.000,C 90.000,E1 24.823} C_DIS
LIN {X 0.231,Y -549.827,Z 1398.933,A 0.000,B 0.000,C 90.000,E1 23.951} C_DIS
LIN {X 0.133,Y -544.356,Z 1398.929,A 0.000,B 0.000,C 90.000,E1 23.259} C_DIS
LIN {X 0.003,Y -536.229,Z 1398.924,A 0.000,B 0.000,C 90.000,E1 22.280} C_DIS
LIN {X -0.025,Y -526.121,Z 1398.918,A 0.000,B 0.000,C 90.000,E1 21.153} C_DIS
LIN {X 0.208,Y -515.677,Z 1398.911,A 0.000,B 0.000,C 90.000,E1 19.993} C_DIS
LIN {X -0.094,Y -508.842,Z 1398.907,A 0.000,B 0.000,C 90.000,E1 19.322} C_DIS
LIN {X -0.216,Y -499.261,Z 1398.902,A 0.000,B 0.000,C 90.000,E1 18.362} C_DIS
LIN {X 0.083,Y -489.643,Z 1398.896,A 0.000,B 0.000,C 90.000,E1 17.347} C_DIS
LIN {X -0.073,Y -477.222,Z 1398.889,A 0.000,B 0.000,C 90.000,E1 16.079} C_DIS
LIN {X 0.143,Y -460.665,Z 1398.880,A 0.000,B 0.000,C 90.000,E1 14.300} C_DIS
LIN {X -0.029,Y -446.775,Z 1398.871,A 0.000,B 0.000,C 90.000,E1 12.827} C_DIS
LIN {X 0.106,Y -438.401,Z 1398.866,A 0.000,B 0.000,C 90.000,E1 11.883} C_DIS
LIN {X 0.114,Y -430.134,Z 1398.861,A 0.000,B 0.000,C 90.000,E1 10.950} C_DIS
LIN {X 0.138,Y -413.885,Z 1398.850,A 0.000,B 0.000,C 90.000,E1 8.973} C_DIS
LIN {X -0.027,Y -401.745,Z 1398.842,A 0.000,B 0.000,C 90.000,E1 7.466} C_DIS
LIN {X -0.066,Y -393.584,Z 1398.836,A 0.000,B 0.000,C 90.000,E1 6.429} C_DIS
LIN {X -0.185,Y -389.024,Z 1398.832,A 0.000,B 0.000,C 90.000,E1 5.739} C_DIS
LIN {X -0.150,Y -388.639,Z 1398.831,A 0.000,B 0.000,C 90.000,E1 5.625} C_DIS
LIN {X -0.188,Y -388.627,Z 1398.831,A 0.000,B 0.000,C 90.000,E1 5.625} C_DIS
LIN {X 0.072,Y -388.953,Z 1398.830,A 0.000,B 0.000,C 90.000,E1 5.391} C_DIS
LIN {X 0.035,Y -388.969,Z 1398.830,A 0.000,B 0.000,C 90.000,E1 5.391} C_DIS
LIN {X -0.107,Y -393.064,Z 1398.827,A 0.000,B 0.000,C 90.000,E1 4.935} C_DIS
LIN {X 0.135,Y -401.609,Z 1398.823,A 0.000,B 0.000,C 90.000,E1 4.131} C_DIS
LIN {X -0.034,Y -405.954,Z 1398.821,A 0.000,B 0.000,C 90.000,E1 3.726} C_DIS
LIN {X -0.195,Y -410.062,Z 1398.818,A 0.000,B 0.000,C 90.000,E1 3.269} C_DIS
LIN {X -0.115,Y -413.356,Z 1398.816,A 0.000,B 0.000,C 90.000,E1 2.865} C_DIS
LIN {X -0.025,Y -417.114,Z 1398.813,A 0.000,B 0.000,C 90.000,E1 2.350} C_DIS
LIN {X 0.003,Y -420.686,Z 1398.810,A 0.000,B 0.000,C 90.000,E1 1.835} C_DIS
LIN {X 0.137,Y -427.181,Z 1398.805,A 0.000,B 0.000,C 90.000,E1 0.802} C_DIS
LIN {X 0.000,Y -432.240,Z 1398.800,A 0.000,B 0.000,C 90.000,E1 360.000} C_DIS
LIN {X -0.094,Y -437.322,Z 1398.795,A 0.000,B 0.000,C 90.000,E1 359.141} C_DIS
LIN {X 0.173,Y -441.978,Z 1398.791,A 0.000,B 0.000,C 90.000,E1 358.282} C_DIS
LIN {X -0.007,Y -445.460,Z 1398.787,A 0.000,B 0.000,C 90.000,E1 357.650} C_DIS
LIN {X 0.195,Y -447.562,Z 1398.784,A 0.000,B 0.000,C 90.000,E1 357.135} C_DIS
LIN {X -0.087,Y -448.727,Z 1398.782,A 0.000,B 0.000,C 90.000,E1 356.846} C_DIS
LIN {X 0.058,Y -449.653,Z 1398.781,A 0.000,B 0.000,C 90.000,E1 356.502} C_DIS
LIN {X 0.206,Y -450.262,Z 1398.779,A 0.000,B 0.000,C 90.000,E1 356.159} C_DIS
LIN {X -0.061,Y -450.242,Z 1398.777,A 0.000,B 0.000,C 90.000,E1 355.869} C_DIS
LIN {X 0.203,Y -449.757,Z 1398.776,A 0.000,B 0.000,C 90.000,E1 355.698} C_DIS
LIN {X -0.028,Y -448.958,Z 1398.776,A 0.000,B 0.000,C 90.000,E1 355.641} C_DIS
LIN {X 0.031,Y -446.835,Z 1398.776,A 0.000,B 0.000,C 90.000,E1 355.584} C_DIS
LIN {X 0.108,Y -390.773,Z 1398.772,A 0.000,B 0.000,C 90.000,E1 354.951} C_DIS
LIN {X -0.057,Y -359.452,Z 1398.770,A 0.000,B 0.000,C 90.000,E1 354.546} C_DIS
LIN {X -0.082,Y -359.426,Z 1398.770,A 0.000,B 0.000,C 90.000,E1 354.546} C_DIS
LIN {X 0.147,Y -359.026,Z 1398.762,A 0.000,B 0.000,C 90.000,E1 353.166} C_DIS
LIN {X -0.180,Y -359.493,Z 1398.727,A 0.000,B 0.000,C 90.000,E1 346.825} C_DIS
LIN {X -0.013,Y -359.545,Z 1398.723,A 0.000,B 0.000,C 90.000,E1 346.047} C_DIS
LIN {X 0.092,Y -361.953,Z 1398.683,A 0.000,B 0.000,C 90.000,E1 338.901} C_DIS
LIN {X 0.108,Y -366.176,Z 1398.641,A 0.000,B 0.000,C 90.000,E1 331.435} C_DIS
LIN {X 0.133,Y -371.179,Z 1398.604,A 0.000,B 0.000,C 90.000,E1 324.769} C_DIS
LIN {X 0.120,Y -371.611,Z 1398.602,A 0.000,B 0.000,C 90.000,E1 324.402} C_DIS
LIN {X 0.167,Y -373.689,Z 1398.586,A 0.000,B 0.000,C 90.000,E1 321.457} C_DIS
LIN {X -0.066,Y -378.114,Z 1398.564,A 0.000,B 0.000,C 90.000,E1 317.472} C_DIS
LIN {X -0.046,Y -384.228,Z 1398.530,A 0.000,B 0.000,C 90.000,E1 311.310} C_DIS
LIN {X -0.002,Y -384.732,Z 1398.527,A 0.000,B 0.000,C 90.000,E1 310.943} C_DIS
LIN {X 0.243,Y -390.898,Z 1398.494,A 0.000,B 0.000,C 90.000,E1 304.818} C_DIS
LIN {X 0.088,Y -391.342,Z 1398.492,A 0.000,B 0.000,C 90.000,E1 304.485} C_DIS
LIN {X -0.090,Y -397.053,Z 1398.458,A 0.000,B 0.000,C 90.000,E1 298.487} C_DIS
LIN {X 0.216,Y -401.443,Z 1398.427,A 0.000,B 0.000,C 90.000,E1 292.823} C_DIS
LIN {X -0.074,Y -401.675,Z 1398.425,A 0.000,B 0.000,C 90.000,E1 292.514} C_DIS
LIN {X -0.044,Y -404.531,Z 1398.396,A 0.000,B 0.000,C 90.000,E1 287.275} C_DIS
LIN {X 0.057,Y -404.763,Z 1398.394,A 0.000,B 0.000,C 90.000,E1 286.913} C_DIS
LIN {X -0.037,Y -406.152,Z 1398.363,A 0.000,B 0.000,C 90.000,E1 281.366} C_DIS
LIN {X 0.067,Y -405.646,Z 1398.334,A 0.000,B 0.000,C 90.000,E1 276.144} C_DIS
LIN {X 0.072,Y -405.630,Z 1398.332,A 0.000,B 0.000,C 90.000,E1 275.796} C_DIS
LIN {X 0.145,Y -403.555,Z 1398.305,A 0.000,B 0.000,C 90.000,E1 270.917} C_DIS
LIN {X 0.080,Y -403.084,Z 1398.301,A 0.000,B 0.000,C 90.000,E1 270.229} C_DIS
LIN {X -0.094,Y -399.028,Z 1398.272,A 0.000,B 0.000,C 90.000,E1 265.008} C_DIS
LIN {X -0.176,Y -398.159,Z 1398.268,A 0.000,B 0.000,C 90.000,E1 264.318} C_DIS
LIN {X 0.077,Y -392.952,Z 1398.241,A 0.000,B 0.000,C 90.000,E1 259.342} C_DIS
LIN {X 0.035,Y -392.522,Z 1398.239,A 0.000,B 0.000,C 90.000,E1 258.993} C_DIS
LIN {X 0.182,Y -386.150,Z 1398.213,A 0.000,B 0.000,C 90.000,E1 254.338} C_DIS
LIN {X 0.142,Y -385.033,Z 1398.207,A 0.000,B 0.000,C 90.000,E1 253.268} C_DIS
LIN {X 0.015,Y -378.167,Z 1398.183,A 0.000,B 0.000,C 90.000,E1 248.954} C_DIS
LIN {X 0.229,Y -375.932,Z 1398.173,A 0.000,B 0.000,C 90.000,E1 247.102} C_DIS
LIN {X -0.152,Y -369.142,Z 1398.151,A 0.000,B 0.000,C 90.000,E1 243.127} C_DIS
LIN {X 0.077,Y -366.291,Z 1398.138,A 0.000,B 0.000,C 90.000,E1 240.873} C_DIS
LIN {X 0.152,Y -358.377,Z 1398.111,A 0.000,B 0.000,C 90.000,E1 236.008} C_DIS
LIN {X -0.006,Y -356.073,Z 1398.101,A 0.000,B 0.000,C 90.000,E1 234.149} C_DIS
LIN {X -0.066,Y -348.512,Z 1398.073,A 0.000,B 0.000,C 90.000,E1 229.218} C_DIS
LIN {X 0.006,Y -345.938,Z 1398.061,A 0.000,B 0.000,C 90.000,E1 226.905} C_DIS
LIN {X -0.029,Y -339.152,Z 1398.033,A 0.000,B 0.000,C 90.000,E1 221.881} C_DIS
LIN {X -0.167,Y -336.979,Z 1398.020,A 0.000,B 0.000,C 90.000,E1 219.564} C_DIS
LIN {X -0.125,Y -335.494,Z 1398.013,A 0.000,B 0.000,C 90.000,E1 218.382} C_DIS
LIN {X -0.112,Y -329.854,Z 1397.980,A 0.000,B 0.000,C 90.000,E1 212.467} C_DIS
LIN {X -0.004,Y -329.095,Z 1397.974,A 0.000,B 0.000,C 90.000,E1 211.258} C_DIS
LIN {X -0.125,Y -324.392,Z 1397.938,A 0.000,B 0.000,C 90.000,E1 204.899} C_DIS
LIN {X 0.087,Y -323.877,Z 1397.929,A 0.000,B 0.000,C 90.000,E1 203.259} C_DIS
LIN {X 0.063,Y -323.404,Z 1397.925,A 0.000,B 0.000,C 90.000,E1 202.461} C_DIS
LIN {X -0.021,Y -321.132,Z 1397.880,A 0.000,B 0.000,C 90.000,E1 194.426} C_DIS
LIN {X 0.141,Y -321.187,Z 1397.837,A 0.000,B 0.000,C 90.000,E1 186.606} C_DIS
LIN {X 0.113,Y -321.342,Z 1397.837,A 0.000,B 0.000,C 90.000,E1 186.606} C_DIS
LIN {X 0.093,Y -360.465,Z 1397.833,A 0.000,B 0.000,C 90.000,E1 185.910} C_DIS
LIN {X -0.154,Y -407.540,Z 1397.829,A 0.000,B 0.000,C 90.000,E1 185.277} C_DIS
LIN {X -0.116,Y -416.320,Z 1397.829,A 0.000,B 0.000,C 90.000,E1 185.163} C_DIS
LIN {X -0.086,Y -418.194,Z 1397.828,A 0.000,B 0.000,C 90.000,E1 185.106} C_DIS
LIN {X 0.002,Y -419.060,Z 1397.828,A 0.000,B 0.000,C 90.000,E1 184.992} C_DIS
LIN {X 0.134,Y -419.939,Z 1397.826,A 0.000,B 0.000,C 90.000,E1 184.645} C_DIS
LIN {X 0.157,Y -419.996,Z 1397.824,A 0.000,B 0.000,C 90.000,E1 184.302} C_DIS
LIN {X 0.213,Y -419.684,Z 1397.822,A 0.000,B 0.000,C 90.000,E1 183.955} C_DIS
LIN {X -0.149,Y -418.570,Z 1397.818,A 0.000,B 0.000,C 90.000,E1 183.326} C_DIS
LIN {X -0.075,Y -417.263,Z 1397.815,A 0.000,B 0.000,C 90.000,E1 182.636} C_DIS
LIN {X -0.030,Y -415.878,Z 1397.811,A 0.000,B 0.000,C 90.000,E1 181.949} C_DIS
LIN {X 0.017,Y -414.312,Z 1397.807,A 0.000,B 0.000,C 90.000,E1 181.260} C_DIS
LIN {X 0.047,Y -411.488,Z 1397.801,A 0.000,B 0.000,C 90.000,E1 180.229} C_DIS
LIN {X 0.049,Y -409.301,Z 1397.797,A 0.000,B 0.000,C 90.000,E1 179.542} C_DIS
LIN {X 0.018,Y -405.630,Z 1397.792,A 0.000,B 0.000,C 90.000,E1 178.511} C_DIS
LIN {X -0.052,Y -401.160,Z 1397.786,A 0.000,B 0.000,C 90.000,E1 177.478} C_DIS
LIN {X -0.120,Y -397.745,Z 1397.782,A 0.000,B 0.000,C 90.000,E1 176.788} C_DIS
LIN {X 0.147,Y -392.897,Z 1397.777,A 0.000,B 0.000,C 90.000,E1 175.869} C_DIS
LIN {X -0.128,Y -385.382,Z 1397.770,A 0.000,B 0.000,C 90.000,E1 174.666} C_DIS
LIN {X 0.102,Y -381.025,Z 1397.766,A 0.000,B 0.000,C 90.000,E1 173.913} C_DIS
LIN {X -0.124,Y -371.161,Z 1397.756,A 0.000,B 0.000,C 90.000,E1 172.129} C_DIS
LIN {X 0.169,Y -364.888,Z 1397.749,A 0.000,B 0.000,C 90.000,E1 170.792} C_DIS
LIN {X -0.082,Y -362.440,Z 1397.746,A 0.000,B 0.000,C 90.000,E1 170.274} C_DIS
LIN {X 0.181,Y -361.130,Z 1397.744,A 0.000,B 0.000,C 90.000,E1 169.859} C_DIS
LIN {X -0.143,Y -359.074,Z 1397.740,A 0.000,B 0.000,C 90.000,E1 169.162} C_DIS
LIN {X 0.084,Y -358.937,Z 1397.739,A 0.000,B 0.000,C 90.000,E1 169.050} C_DIS
LIN {X 0.047,Y -358.935,Z 1397.739,A 0.000,B 0.000,C 90.000,E1 169.050} C_DIS
LIN {X 0.116,Y -359.716,Z 1397.737,A 0.000,B 0.000,C 90.000,E1 168.634} C_DIS
LIN {X 0.079,Y -359.735,Z 1397.737,A 0.000,B 0.000,C 90.000,E1 168.634} C_DIS
LIN {X 0.124,Y -363.546,Z 1397.733,A 0.000,B 0.000,C 90.000,E1 167.993} C_DIS
LIN {X 0.167,Y -367.598,Z 1397.730,A 0.000,B 0.000,C 90.000,E1 167.409} C_DIS
LIN {X 0.150,Y -375.749,Z 1397.725,A 0.000,B 0.000,C 90.000,E1 166.408} C_DIS
LIN {X 0.084,Y -387.724,Z 1397.717,A 0.000,B 0.000,C 90.000,E1 165.102} C_DIS
LIN {X 0.140,Y -399.980,Z 1397.711,A 0.000,B 0.000,C 90.000,E1 163.866} C_DIS
LIN {X -0.207,Y -415.384,Z 1397.703,A 0.000,B 0.000,C 90.000,E1 162.543} C_DIS
LIN {X -0.134,Y -435.936,Z 1397.694,A 0.000,B 0.000,C 90.000,E1 160.859} C_DIS
LIN {X 0.126,Y -446.895,Z 1397.689,A 0.000,B 0.000,C 90.000,E1 159.953} C_DIS
LIN {X 0.074,Y -454.678,Z 1397.685,A 0.000,B 0.000,C 90.000,E1 159.337} C_DIS
LIN {X -0.014,Y -465.419,Z 1397.680,A 0.000,B 0.000,C 90.000,E1 158.465} C_DIS
LIN {X -0.156,Y -472.849,Z 1397.677,A 0.000,B 0.000,C 90.000,E1 157.847} C_DIS
LIN {X -0.006,Y -478.646,Z 1397.674,A 0.000,B 0.000,C 90.000,E1 157.305} C_DIS
LIN {X 0.019,Y -490.153,Z 1397.668,A 0.000,B 0.000,C 90.000,E1 156.230} C_DIS
LIN {X 0.215,Y -495.756,Z 1397.665,A 0.000,B 0.000,C 90.000,E1 155.665} C_DIS
LIN {X -0.157,Y -501.225,Z 1397.662,A 0.000,B 0.000,C 90.000,E1 155.153} C_DIS
LIN {X -0.043,Y -505.220,Z 1397.660,A 0.000,B 0.000,C 90.000,E1 154.717} C_DIS
LIN {X -0.259,Y -511.627,Z 1397.656,A 0.000,B 0.000,C 90.000,E1 154.024} C_DIS
LIN {X 0.046,Y -515.246,Z 1397.653,A 0.000,B 0.000,C 90.000,E1 153.563} C_DIS
LIN {X -0.047,Y -522.249,Z 1397.648,A 0.000,B 0.000,C 90.000,E1 152.692} C_DIS
LIN {X 0.015,Y -526.441,Z 1397.645,A 0.000,B 0.000,C 90.000,E1 152.103} C_DIS
LIN {X -0.041,Y -531.049,Z 1397.641,A 0.000,B 0.000,C 90.000,E1 151.385} C_DIS
LIN {X 0.090,Y -534.311,Z 1397.638,A 0.000,B 0.000,C 90.000,E1 150.795} C_DIS
LIN {X -0.221,Y -537.080,Z 1397.635,A 0.000,B 0.000,C 90.000,E1 150.255} C_DIS
LIN {X -0.183,Y -540.069,Z 1397.631,A 0.000,B 0.000,C 90.000,E1 149.537} C_DIS
LIN {X 0.008,Y -542.170,Z 1397.628,A 0.000,B 0.000,C 90.000,E1 148.948} C_DIS
LIN {X -0.231,Y -544.947,Z 1397.623,A 0.000,B 0.000,C 90.000,E1 148.122} C_DIS
LIN {X -0.006,Y -546.613,Z 1397.620,A 0.000,B 0.000,C 90.000,E1 147.533} C_DIS
LIN {X -0.195,Y -548.663,Z 1397.615,A 0.000,B 0.000,C 90.000,E1 146.707} C_DIS
LIN {X -0.361,Y -550.434,Z 1397.610,A 0.000,B 0.000,C 90.000,E1 145.881} C_DIS
LIN {X 0.201,Y -551.452,Z 1397.607,A 0.000,B 0.000,C 90.000,E1 145.261} C_DIS
LIN {X 0.319,Y -552.366,Z 1397.604,A 0.000,B 0.000,C 90.000,E1 144.689} C_DIS
LIN {X -0.259,Y -553.327,Z 1397.599,A 0.000,B 0.000,C 90.000,E1 143.909} C_DIS
LIN {X 0.090,Y -554.676,Z 1397.592,A 0.000,B 0.000,C 90.000,E1 142.477} C_DIS
LIN {X 0.098,Y -556.083,Z 1397.582,A 0.000,B 0.000,C 90.000,E1 140.803} C_DIS
LIN {X -0.030,Y -556.972,Z 1397.576,A 0.000,B 0.000,C 90.000,E1 139.703} C_DIS
LIN {X -0.133,Y -557.734,Z 1397.568,A 0.000,B 0.000,C 90.000,E1 138.324} C_DIS
LIN {X -0.293,Y -558.251,Z 1397.562,A 0.000,B 0.000,C 90.000,E1 137.229} C_DIS
LIN {X 0.130,Y -559.036,Z 1397.552,A 0.000,B 0.000,C 90.000,E1 135.243} C_DIS
LIN {X -0.024,Y -559.360,Z 1397.545,A 0.000,B 0.000,C 90.000,E1 134.150} C_DIS
LIN {X -0.092,Y -559.717,Z 1397.538,A 0.000,B 0.000,C 90.000,E1 132.771} C_DIS
LIN {X -0.226,Y -559.915,Z 1397.531,A 0.000,B 0.000,C 90.000,E1 131.676} C_DIS
LIN {X -0.101,Y -560.177,Z 1397.521,A 0.000,B 0.000,C 90.000,E1 129.725} C_DIS
LIN {X -0.324,Y -560.681,Z 1397.510,A 0.000,B 0.000,C 90.000,E1 127.810} C_DIS
LIN {X -0.055,Y -561.195,Z 1397.493,A 0.000,B 0.000,C 90.000,E1 124.739} C_DIS
LIN {X 0.038,Y -561.499,Z 1397.491,A 0.000,B 0.000,C 90.000,E1 124.452} C_DIS
LIN {X 0.005,Y -562.045,Z 1397.487,A 0.000,B 0.000,C 90.000,E1 123.627} C_DIS
LIN {X -0.210,Y -562.552,Z 1397.485,A 0.000,B 0.000,C 90.000,E1 123.372} C_DIS
LIN {X 0.225,Y -563.683,Z 1397.484,A 0.000,B 0.000,C 90.000,E1 123.086} C_DIS
LIN {X 0.090,Y -564.819,Z 1397.484,A 0.000,B 0.000,C 90.000,E1 123.007} C_DIS
LIN {X -0.013,Y -566.186,Z 1397.483,A 0.000,B 0.000,C 90.000,E1 122.959} C_DIS
LIN {X -0.075,Y -572.261,Z 1397.482,A 0.000,B 0.000,C 90.000,E1 122.801} C_DIS
LIN {X 0.056,Y -578.128,Z 1397.482,A 0.000,B 0.000,C 90.000,E1 122.673} C_DIS
LIN {X -0.147,Y -580.851,Z 1397.481,A 0.000,B 0.000,C 90.000,E1 122.625} C_DIS
LIN {X -0.255,Y -583.671,Z 1397.481,A 0.000,B 0.000,C 90.000,E1 122.546} C_DIS
LIN {X -0.094,Y -586.470,Z 1397.480,A 0.000,B 0.000,C 90.000,E1 122.418} C_DIS
LIN {X 0.130,Y -589.449,Z 1397.479,A 0.000,B 0.000,C 90.000,E1 122.260} C_DIS
LIN {X -0.132,Y -592.321,Z 1397.479,A 0.000,B 0.000,C 90.000,E1 122.133} C_DIS
LIN {X -0.259,Y -596.641,Z 1397.477,A 0.000,B 0.000,C 90.000,E1 121.878} C_DIS
LIN {X 0.079,Y -600.838,Z 1397.475,A 0.000,B 0.000,C 90.000,E1 121.544} C_DIS
LIN {X -0.237,Y -606.421,Z 1397.473,A 0.000,B 0.000,C 90.000,E1 121.131} C_DIS
LIN {X -0.317,Y -611.614,Z 1397.470,A 0.000,B 0.000,C 90.000,E1 120.669} C_DIS
LIN {X 0.128,Y -616.324,Z 1397.468,A 0.000,B 0.000,C 90.000,E1 120.129} C_DIS
LIN {X 0.086,Y -620.697,Z 1397.465,A 0.000,B 0.000,C 90.000,E1 119.617} C_DIS
LIN {X -0.166,Y -624.494,Z 1397.462,A 0.000,B 0.000,C 90.000,E1 119.127} C_DIS
LIN {X -0.147,Y -628.720,Z 1397.458,A 0.000,B 0.000,C 90.000,E1 118.487} C_DIS
LIN {X -0.088,Y -632.105,Z 1397.455,A 0.000,B 0.000,C 90.000,E1 117.847} C_DIS
LIN {X -0.055,Y -633.270,Z 1397.453,A 0.000,B 0.000,C 90.000,E1 117.590} C_DIS
LIN {X 0.020,Y -635.170,Z 1397.450,A 0.000,B 0.000,C 90.000,E1 117.078} C_DIS
LIN {X 0.064,Y -635.788,Z 1397.449,A 0.000,B 0.000,C 90.000,E1 116.821} C_DIS
LIN {X 0.210,Y -636.639,Z 1397.445,A 0.000,B 0.000,C 90.000,E1 116.052} C_DIS
LIN {X -0.262,Y -636.366,Z 1397.442,A 0.000,B 0.000,C 90.000,E1 115.591} C_DIS
LIN {X -0.212,Y -635.966,Z 1397.441,A 0.000,B 0.000,C 90.000,E1 115.335} C_DIS
LIN {X -0.117,Y -634.678,Z 1397.438,A 0.000,B 0.000,C 90.000,E1 114.823} C_DIS
LIN {X -0.096,Y -633.977,Z 1397.437,A 0.000,B 0.000,C 90.000,E1 114.695} C_DIS
LIN {X -0.317,Y -632.265,Z 1397.436,A 0.000,B 0.000,C 90.000,E1 114.463} C_DIS
LIN {X -0.280,Y -630.710,Z 1397.434,A 0.000,B 0.000,C 90.000,E1 114.207} C_DIS
LIN {X 0.146,Y -625.130,Z 1397.432,A 0.000,B 0.000,C 90.000,E1 113.695} C_DIS
LIN {X 0.065,Y -623.321,Z 1397.431,A 0.000,B 0.000,C 90.000,E1 113.590} C_DIS
LIN {X -0.146,Y -620.923,Z 1397.431,A 0.000,B 0.000,C 90.000,E1 113.515} C_DIS
LIN {X 0.210,Y -619.056,Z 1397.430,A 0.000,B 0.000,C 90.000,E1 113.387} C_DIS
LIN {X 0.201,Y -616.904,Z 1397.429,A 0.000,B 0.000,C 90.000,E1 113.259} C_DIS
LIN {X -0.230,Y -614.601,Z 1397.429,A 0.000,B 0.000,C 90.000,E1 113.206} C_DIS
LIN {X -0.069,Y -609.120,Z 1397.428,A 0.000,B 0.000,C 90.000,E1 113.003} C_DIS
LIN {X -0.132,Y -606.335,Z 1397.427,A 0.000,B 0.000,C 90.000,E1 112.898} C_DIS
LIN {X -0.089,Y -598.528,Z 1397.426,A 0.000,B 0.000,C 90.000,E1 112.642} C_DIS
LIN {X 0.113,Y -597.850,Z 1397.426,A 0.000,B 0.000,C 90.000,E1 112.589} C_DIS
LIN {X 0.077,Y -597.792,Z 1397.426,A 0.000,B 0.000,C 90.000,E1 112.589} C_DIS
LIN {X -0.215,Y -607.440,Z 1397.422,A 0.000,B 0.000,C 90.000,E1 111.897} C_DIS
LIN {X -0.087,Y -614.150,Z 1397.419,A 0.000,B 0.000,C 90.000,E1 111.334} C_DIS
LIN {X 0.097,Y -618.148,Z 1397.417,A 0.000,B 0.000,C 90.000,E1 110.972} C_DIS
LIN {X 0.215,Y -623.109,Z 1397.414,A 0.000,B 0.000,C 90.000,E1 110.482} C_DIS
LIN {X 0.122,Y -627.895,Z 1397.411,A 0.000,B 0.000,C 90.000,E1 109.993} C_DIS
LIN {X -0.284,Y -633.105,Z 1397.408,A 0.000,B 0.000,C 90.000,E1 109.396} C_DIS
LIN {X 0.139,Y -636.925,Z 1397.405,A 0.000,B 0.000,C 90.000,E1 108.852} C_DIS
LIN {X -0.185,Y -641.868,Z 1397.401,A 0.000,B 0.000,C 90.000,E1 108.127} C_DIS
LIN {X 0.150,Y -646.002,Z 1397.396,A 0.000,B 0.000,C 90.000,E1 107.347} C_DIS
LIN {X 0.068,Y -648.608,Z 1397.393,A 0.000,B 0.000,C 90.000,E1 106.732} C_DIS
LIN {X -0.212,Y -650.168,Z 1397.390,A 0.000,B 0.000,C 90.000,E1 106.260} C_DIS
LIN {X -0.346,Y -650.902,Z 1397.389,A 0.000,B 0.000,C 90.000,E1 106.024} C_DIS
LIN {X 0.069,Y -652.338,Z 1397.385,A 0.000,B 0.000,C 90.000,E1 105.245} C_DIS
LIN {X -0.303,Y -653.372,Z 1397.381,A 0.000,B 0.000,C 90.000,E1 104.537} C_DIS
